// ---- 04_Application/OPC/OpcUa.TcPOU
PROGRAM OpcUa
///////////////////
// OPC UA Management 
// Commands are resetted to FALSE right after being received . Protection against rapide consecutives commands . Protection against simultaneous commands.
///////////////////
VAR_INPUT PERSISTENT
	ParamTimeOutTc			: TIME:=T#1S;		(* (s)Minimum duration before two consecutives commands *)
	ParamNbCmdBlock			: UINT  := 1 ; 		(* Number of commands per block. Commands in the same block can not be executed in the same time. *)
//Test
END_VAR             		
                    		
                    		
VAR_INPUT           		
                    		
    {attribute 'OPC.UA.DA' := '1'}                		
	AllDataR 				: AllDataR; // All Data Read Only
	
	{attribute 'OPC.UA.DA' := '1'}                		
	AllDataWPulse 			: AllDataWPulse; //  All boolean OPC UA to be written  that will be converted to tap by resetting the entry to false after two seconds. 
	
	AllDataWToggle 			: AllDataWToggle; // All boolean OPC UA to be written as a toggle
    
    {attribute 'OPC.UA.DA' := '1'}            		
	AllValueW 				: AllValueW; // All non boolean OPC UA data to be  written 
	                		
	AllRtc					: AllDataWPulse;	// OUtput of the AllDataWPulse . 
	
	// Test Mise à jour Parameters via OPC UA
	
	//AllDataParameterWrite	: AllDataParameter;	// Structure qui permet d'écrire les valeurs des paramètres via OPC UA
   		
END_VAR             		
VAR                 		
//	Buffer_AllW				: ARRAY[1..500] OF BOOL ;      
	Buffer_TcWord			: ARRAY[1..500] OF BOOL ;  
	Buffer_Rtc   			: ARRAY[1..500] OF BOOL ;  
	
	CP_TcAllow				: BOOL; // The power plan can received TC

	bInit					: BOOL;
	TempoTcRunning			: TON;
	                		
	// M_TC //      		
	TcIsRunning				: BOOL;
	NbTcAskedBlock			: BYTE;	    
	bTooManyCmd				: BOOL;		// At least one block has too many simultaneous commands. 
	bAtLeastOne				: BOOL;     // There is at least one commAND                              
	                        
	// M_ACKNOWLEDGE        
	F_Tap_OPC				: ARRAY[1..23] OF FB_TapVariable ; 
	F_Tap_OPC_SUB_MV		: ARRAY[1..16] OF FB_TapVariable ; 
	F_Tap_OPC_PTR			: ARRAY[1..CstNbPTR_G] OF ARRAY[1..6] OF FB_TapVariable ;		
	F_Tap_OPC_Inv			: ARRAY[1..CstNbPTR_G] OF ARRAY[1..CstNbInv_PTR_G] OF ARRAY[1..4] OF FB_TapVariable ;		
	F_Tap_OPC_GRID			: ARRAY[1..10] OF FB_TapVariable ; 
	F_Tap_OPC_PP			: ARRAY[1..10] OF FB_TapVariable ;	
	F_Tap_OPC_SUB_MV_InhibRead		: ARRAY[1..10] OF FB_TapVariable ;	
	
	
	F_Tap_OPC_INV_InhibRead : ARRAY[1..CstNbPTR_G] OF ARRAY[1..CstNbInv_PTR_G] OF FB_TapVariable ;	
	F_Tap_OPC_SL_InhibRead : ARRAY[1..CstNbPTR_G] OF FB_TapVariable ;	

	F_Tap_Inhib : ARRAY[1..1000] OF FB_TapVariable ;	
	
	
	Test_SmS_Rtrig			: R_TRIG ; 
	Rtrig_StayConnect		: R_TRIG;
	Rtrig_IpLauncher		: R_TRIG;
	Rtrig_HHCollector		: R_TRIG;
	Rtrig_RestartPlc		: R_TRIG;
	R_TRIGTanPhi			: R_TRIG ; 
	R_TRIG_InhibIO			: R_TRIG;
	bReadFromTargetInfos	: BOOL ; 
	// Intermediary commands
	PP_SetptP_Old							: REAL;
	PP_SetptQ_Old							: REAL;
	

	
END_VAR


VAR
	// WAGO Variable transcription
	OpcUaServer_1 : REAL ; 
	OpcUaServer_2 : REAL ; 
	OpcUaServer_3 : REAL ; 
	OpcUaServer_4 : REAL ; 
	OpcUaServer_5 : REAL ; 
	OpcUaServer_6 : REAL ; 
	OpcUaServer_7 : REAL ; 
	OpcUaServer_8 : REAL ; 
	OpcUaServer_9 : REAL ; 
	OpcUaServer_10 : REAL ; 
	OpcUaServer_11 : REAL ; 
	OpcUaServer_12 : REAL ; 
	OpcUaServer_13 : REAL ; 
	OpcUaServer_14 : REAL ; 
	OpcUaServer_15 : REAL ; 
	OpcUaServer_16 : REAL ; 
	OpcUaServer_17 : REAL ; 
	OpcUaServer_18 : REAL ; 
	OpcUaServer_19 : REAL ; 
	OpcUaServer_20 : REAL ; 
	OpcUaServer_21 : REAL ; 
	OpcUaServer_22 : REAL ; 
	OpcUaServer_23 : REAL ; 
	OpcUaServer_24 : REAL ; 
	OpcUaServer_25 : REAL ; 
	OpcUaServer_26 : REAL ; 
	OpcUaServer_27 : REAL ; 
	OpcUaServer_28 : REAL ; 
	OpcUaServer_29 : REAL ; 
	OpcUaServer_30 : REAL ; 
	OpcUaServer_31 : REAL ; 
	OpcUaServer_32 : REAL ; 
	OpcUaServer_33 : REAL ; 
	OpcUaServer_34 : REAL ; 
	OpcUaServer_35 : REAL ; 
	OpcUaServer_36 : REAL ; 
	OpcUaServer_37 : REAL ; 
	OpcUaServer_38 : REAL ; 
	OpcUaServer_39 : REAL ; 
	OpcUaServer_40 : REAL ; 
	OpcUaServer_41 : REAL ; 
	OpcUaServer_42 : REAL ; 
	OpcUaServer_43 : REAL ; 

END_VAR

	IF NOT bInit THEN
		M_Init() ; 
		bInit		:= TRUE ; 
	ELSE
		CP_TcAllow := TRUE;
		M_Evaluate();
		M_TC();
		M_Acknowledge();
		M_InhibAllowAll() ; 
		//M_Wago()
	END_IF

METHOD M_Acknowledge : BOOL
VAR
		KK: INT;
		LL: INT;
	JJ: UINT;
	TapTrigger: BOOL;
END_VAR


// 					ATTENTION				//
// Utiliser le AllRtc et pas le AllDataR 	//

	
// Defaults Actions
	// Reset SMS Server
	F_Tap_OPC[2](TapTrigger:= AllRtc.CmdReset_ServerSMS , TapOut := SMS_Server.IN_Reset_SmsServer) ; 
	// Delete all SMS
	F_Tap_OPC[3](TapTrigger:= AllRtc.CmdDeleteAllSms , TapOut := SMS_Server.IN_CmdDeleteAllSms) ; 
	// Update SMS & Mail Informations
	F_Tap_OPC[4](TapTrigger:= AllRtc.CmdChangeInfos_PhoneEmail , TapOut := SMS_Server.IN_ChangePhoneMailInfos_OPC) ; 
	F_Tap_OPC[5](TapTrigger:= AllRtc.CmdChangeInfos_PhoneEmail , TapOut := FUN_SendMail.IN_ChangePhoneMailInfos_OPC) ; 
	bReadFromTargetInfos :=	AllRtc.CmdReadInfosFromTarget_PhoneEmail ; 
	// Collect Ip Public
	Rtrig_IpLauncher(CLK:=AllRtc.CmdIpLauncher);
	F_Tap_OPC[6](TapTrigger:= Rtrig_IpLauncher.Q , TapOut := PRG_AnnexesFunctions.IN_bStart_IP) ; 
	
	// Toogle Forced Connect
	Rtrig_StayConnect(CLK:=AllRtc.CmdForcedStay_Connect);
	IF Rtrig_StayConnect.Q THEN
		A1_PP.ParamForcedStayConnect := NOT	A1_PP.ParamForcedStayConnect ;
	END_IF
	// Restart PLC
	//Rtrig_RestartPlc(CLK:=AllRtc.CmdRestart_PLC);
	F_Tap_OPC[8](TapTrigger:= AllRtc.CmdRestart_PLC , TapOut := PRG_AnnexesFunctions.IN_bStart_PLC) ; 
	// Restart Routeur ADSL
	F_Tap_OPC[9](TapTrigger:= AllRtc.CmdReset_Router_ADSL, TapOut := A1_SUBMV.A1_Router_ADSL.IN_CmdRestart) ; 
	//Reset MailServer
	F_Tap_OPC[10](TapTrigger:= AllRtc.CmdReset_ServerMail, TapOut := FUN_SendMail.IN_Reset_OPC) ; 
	// Test sms
	Test_SmS_Rtrig(CLK:=AllRtc.CmdTestSms);
	F_Tap_OPC[11](TapTrigger:= Test_SmS_Rtrig.Q, TapOut := A1_PP.IN_TestMailSms) ; 	
	// Restart Routeur 4G
	F_Tap_OPC[12](TapTrigger:= AllRtc.CmdReset_Router_4G, TapOut := A1_SUBMV.A1_Router_4G.IN_CmdRestart) ;
 	// Restart IPC
	F_Tap_OPC[13](TapTrigger:= AllRtc.CmdReset_IPC, TapOut := A1_SUBMV.A1_IPC.IN_CmdRestart) ;
	
	// Disable sms serveur
	F_Tap_OPC[14](TapTrigger:= AllDataWToggle.CmdStopServer_SMS, TapOut := FUN_Alarms.ParamDisableSMS) ; 
	// Start VPN
	F_Tap_OPC[15](TapTrigger:= AllRtc.CmdStart_Vpn, TapOut := PRG_AnnexesFunctions.IN_bStartVpnConnection) ; 
	// Stop VPN
	F_Tap_OPC[16](TapTrigger:= AllRtc.CmdStop_Vpn, TapOut := PRG_AnnexesFunctions.IN_bStopVpnConnection) ;

	
	
	// Restart Services
	F_Tap_OPC[17](TapTrigger:= AllRtc.CmdRestart_HH 		, TapOut := PRG_AnnexesFunctions.IN_CmdRestart_HH) ; // 1
	F_Tap_OPC[18](TapTrigger:= AllRtc.CmdRestart_OPCUA 		 , TapOut := PRG_AnnexesFunctions.IN_CmdRestart_OPCUA) ; // 
	F_Tap_OPC[19](TapTrigger:= AllRtc.CmdRestart_OpenVPN 	 , TapOut := PRG_AnnexesFunctions.IN_CmdRestart_OpenVPN 	 ) ; // 
	F_Tap_OPC[20](TapTrigger:= AllRtc.CmdRestart_Teamviewer	 , TapOut := PRG_AnnexesFunctions.IN_CmdRestart_Teamviewer) ; // 
	F_Tap_OPC[21](TapTrigger:= AllRtc.CmdRestart_HMIServer 	 , TapOut := PRG_AnnexesFunctions.IN_CmdRestart_HMIServer ) ; // 
	F_Tap_OPC[22](TapTrigger:= AllRtc.CmdRestart_Docker 	 , TapOut := PRG_AnnexesFunctions.IN_CmdRestart_Docker 	  ) ; // 
	F_Tap_OPC[23](TapTrigger:= AllRtc.CmdRestart_Codesys 	 , TapOut := PRG_AnnexesFunctions.IN_CmdRestart_Codesys 	 ) ; // 		
		
	

//SUB_MV
	F_Tap_OPC_SUB_MV[1](TapTrigger:= AllRtc.CmdOpen_MainMVCB , TapOut 	:= A1_SUBMV.IN_CmdOpenMainMVCB) ; 
	F_Tap_OPC_SUB_MV[2](TapTrigger:= AllRtc.CmdClose_MainMVCB , TapOut 	:= A1_SUBMV.IN_CmdCloseMainMVCB) ;
	F_Tap_OPC_SUB_MV[3](TapTrigger:= AllRtc.CmdReset_MainMVCB , TapOut 	:= A1_SUBMV.A1_MainMVCB.IN_CmdReset_L) ; 
	F_Tap_OPC_SUB_MV[4](TapTrigger:= AllRtc.CmdRestart_UPS48 , TapOut 	:= A1_SUBMV.A1_UPS_48v.IN_CmdReStartUPS) ; 	
	
	FOR KK:= 1 TO CstNbFeederMVCB_G DO 
		F_Tap_OPC_SUB_MV[4+(KK-1)*3+1](TapTrigger:= AllRtc.CmdOpen_FeederMVCB[KK] , TapOut := A1_SUBMV.IN_CmdOpenFeederMVCB[KK]) ; 
		F_Tap_OPC_SUB_MV[4+(KK-1)*3+2](TapTrigger:= AllRtc.CmdClose_FeederMVCB[KK] , TapOut := A1_SUBMV.IN_CmdCloseFeederMVCB[KK]) ; 
		F_Tap_OPC_SUB_MV[4+(KK-1)*3+3](TapTrigger:= AllRtc.CmdReset_FeederMVCB[KK] , TapOut := A1_SUBMV.AX_FeederMVCB[KK].IN_CmdReset_L) ; 

	END_FOR 	
	
// PTR 
FOR KK := 1 TO UINT_TO_INT(CstNbPTR_G) DO
	F_Tap_OPC_PTR[KK][1](TapTrigger:= AllRtc.CmdClose_PTR[KK] , TapOut := AX_PTR[KK].A1_MainMVCB_PTR.IN_CmdClose) ;
	F_Tap_OPC_PTR[KK][2](TapTrigger:= AllRtc.CmdOpen_PTR[KK] , TapOut := AX_PTR[KK].A1_MainMVCB_PTR.IN_CmdOpen) ;
	
	FOR JJ:=1 TO CstNbInv_PTR_G DO 
		F_Tap_OPC_Inv[KK][JJ][1](TapTrigger:= AllRtc.CmdStop_INV[KK][JJ] , TapOut := AX_PTR[KK].AX_INV[JJ].IN_CmdStop_Local ) ;
		F_Tap_OPC_Inv[KK][JJ][2](TapTrigger:= AllRtc.CmdStart_INV[KK][JJ] , TapOut := AX_PTR[KK].AX_INV[JJ].IN_CmdStart_Local ) ;		
		
		F_Tap_OPC_Inv[KK][JJ][3](TapTrigger:= AllRtc.CmdToggleCom_Read[KK][JJ] , TapOut := AX_PTR[KK].AX_INV[JJ].IN_CmdToggleRead ) ;
		F_Tap_OPC_Inv[KK][JJ][4](TapTrigger:= AllRtc.CmdToggleCom_Write[KK][JJ] , TapOut := AX_PTR[KK].AX_INV[JJ].IN_CmdToggleWrite ) ;		
	
		
		
		IF AllRtc.CmdStartSetptP_INV[KK][JJ] THEN 
			AX_PTR[KK].AX_INV[JJ].IN_SetptPlimit_Local :=  AllValueW.SetpP_INV[KK][JJ] ; 
		END_IF
		IF AllRtc.CmdStopSetptP_INV[KK][JJ] THEN 
			AX_PTR[KK].AX_INV[JJ].IN_SetptPlimit_Local :=  AX_PTR[KK].AX_INV[JJ].ParamPn ; 
		END_IF
		
	END_FOR
	

	

END_FOR

// DEIE
	F_Tap_OPC_GRID[1](TapTrigger:= AllRtc.CmdAutCpl , TapOut := A1_SUBMV.A1_GRID.IN_CmdAutCpl_other) ; 
	F_Tap_OPC_GRID[2](TapTrigger:= AllRtc.CmdDisconnect , TapOut := A1_SUBMV.A1_GRID.IN_CmdDisconnect_other) ; 
	F_Tap_OPC_GRID[3](TapTrigger:= AllRtc.CmdDisconnect_end , TapOut := A1_SUBMV.A1_GRID.IN_CmdDisconnect_end_other) ; 
	F_Tap_OPC_GRID[4](TapTrigger:= AllRtc.CmdEmergencyDisconnect , TapOut := A1_SUBMV.A1_GRID.IN_CmdEmergencyDisconnect_other) ; 	
	F_Tap_OPC_GRID[5](TapTrigger:= AllRtc.CmdEmergencyDisconnect_end , TapOut := A1_SUBMV.A1_GRID.IN_CmdEmergencyDisconnect_End_other) ; 	
	F_Tap_OPC_GRID[6](TapTrigger:= AllRtc.CmdStartPReg 		, TapOut := A1_SUBMV.A1_GRID.IN_CmdStartPReg_other) ; 
	F_Tap_OPC_GRID[7](TapTrigger:= AllRtc.CmdStopPReg 		, TapOut := A1_SUBMV.A1_GRID.IN_CmdStopPReg_other) ; 
	F_Tap_OPC_GRID[8](TapTrigger:= AllRtc.CmdStartQReg 		, TapOut := A1_SUBMV.A1_GRID.IN_CmdStartQReg_other) ; 
	F_Tap_OPC_GRID[9](TapTrigger:= AllRtc.CmdStopQReg 		, TapOut := A1_SUBMV.A1_GRID.IN_CmdStopQReg_other) ; 


//SUB_MV
	IF AllRtc.CmdStartLocalSetptP_PP THEN
		A1_PP.IN_PIDP_SetptP_local			:=	AllValueW.SetpP_SUB;
		A1_PP.IN_CmdPIDP_LocalMode 	:= TRUE;
	END_IF
	
	IF AllRtc.CmdStopLocalSetptP_PP THEN
		A1_PP.IN_CmdPIDP_LocalMode  	:= FALSE; 
		A1_PP.IN_PIDP_SetptP_local		:= A1_PP.ParamPmax;               
	END_IF
	
	
// PP 
	R_TRIGTanPhi(CLK:= AllRtc.CmdWriteSetptTanPhi ) ; 
	IF R_TRIGTanPhi.Q THEN 
		A1_PP.Param_SetptTanPhi  :=  AllValueW.SetptTanPhi_PP ; 		
	END_IF


//MAIL - SMS 
IF bReadFromTargetInfos THEN 
	AllValueW.AX_MailAddr_OPC		 := AllDataR.MAIL.AX_MailAddr   ; 
	AllValueW.AX_NamesUsers_OPC 	 := AllDataR.MAIL.AX_NomUtili 	; 
	AllValueW.AX_NbPhone_OPC		 := AllDataR.SMS.AX_Numtel 		; 	
	AllValueW.AX_SubscribedMail_OPC  := AllDataR.MAIL.AX_Subscribed ; 	
	AllValueW.AX_SubscribedSms_OPC   := AllDataR.SMS.AX_Subscribed  ; 	
	AllValueW.AX_UserLVL 			 := AllDataR.MAIL.AX_UserLVL    ;  		
	
	bReadFromTargetInfos 			 := FALSE ;
END_IF
END_METHOD

METHOD M_AlarmManagement
//////////////////
// Generates object alarms and manages resets. 
//////////////////

VAR 
	// Method local variables (reinitialized at each cycle) 
	FB_AlarmCodeManager			: FB_AlarmCodeManager ;

	TransfoAlarmCode			: WORD;
	TransfoWarningCode			: WORD;
	ANATempWarningCode			: WORD;    // ANA Temperature Warning Code synthesis 
	ANATempAlarmCode			: WORD;    // ANA Temperature Alarm Code synthesis                               

	AlarmCodeSD_Transfo			: WORD;    // Sd Alarm Code synthesis PTR
	AlarmCodeSD_INV				: WORD;    // Sd Alarm Code synthesis SCADA
	
	VaneWarningCode             : WORD;
	TempSensor_Amb_1WarningCode	: WORD;
	TempSensor_Amb_2WarningCode	: WORD;
	TempSensor_TransfoWarningCode: WORD;

	InvComWarning				: BOOL;		// Aggregated communication warning
	InvComError					: BOOL;		// Aggregated communication Alarm
	InvAlarmCode				: WORD; 
	InvWarningcode				: WORD;
	
	DS_Transfo					: BOOL;
	DS_INV						: BOOL;
END_VAR

	
// ALARM CODE //
	FB_AlarmCodeManager(
		bAlarm1			:= FALSE,//
		bAlarm2			:= FALSE,//
		bAlarm3			:= FALSE,//
		bAlarm4			:= FALSE,//
		bAlarm5			:= FALSE,//
		bAlarm6			:= FALSE,//
		bAlarm7			:= FALSE,//
		bAlarm8			:= FALSE,//
		bAlarm9			:= FALSE,//
		bAlarm10		:= FALSE,//
		bAlarm11		:= FALSE,//
		bAlarm12		:= FALSE,//
		bAlarm13		:= FALSE,//
		bAlarm14		:= FALSE,//
		bAlarm15		:= FALSE,//
		wAlarmCode		=> AllDataR.MesAlarmCode);

// WARNING CODE //
	FB_AlarmCodeManager(
 		bAlarm1			:= CP_TcAllow AND bTooManyCmd AND NOT   TcIsRunning,	// two many action in the same time requested                                 
		bAlarm2			:= bAtLeastOne AND  NOT bTooManyCmd AND NOT CP_TcAllow,  					// Cmd send but the PP do not allow TC
		bAlarm3			:= CP_TcAllow AND bAtLeastOne AND  NOT bTooManyCmd AND   TcIsRunning,		// Wait for previous command to be executed.
		bAlarm4			:= FALSE,//
		bAlarm5			:= FALSE,//
		bAlarm6			:= FALSE,//
		bAlarm7			:= FALSE,//
		bAlarm8			:= FALSE,//
		bAlarm9			:= FALSE,//
		bAlarm10		:= FALSE,//
		bAlarm11		:= FALSE,//
		bAlarm12		:= FALSE,//
		bAlarm13		:= FALSE,//
		bAlarm14		:= FALSE,//
        bAlarm15		:= FALSE,//
		wAlarmCode		=> AllDataR.MesWarningCode);
FB_AlarmCodeManager(
bAlarm1         :=allDataWPulse.CmdReset_ServerSMS,//Reset SMS Server #Interface
bAlarm2         :=allDataWPulse.CmdReset_ServerMail,//Reset Mail server #Interface
bAlarm3         :=allDataWPulse.CmdReset_Router_ADSL,//Restart ADSL router #Interface
bAlarm4         :=allDataWPulse.CmdReset_Router_4G,//Restart 4G router #Interface
bAlarm5         :=allDataWPulse.CmdReset_IPC,//Restart IPC #Interface
bAlarm6         :=allDataWPulse.CmdDeleteAllSms,//Delete all SMS in the buffer #Interface
bAlarm7         :=allDataWPulse.CmdChangeInfos_PhoneEmail,//Apply new changes in MAil and SMS infos #Interface
bAlarm8         :=allDataWPulse.CmdTestSms,//Test SMS function #Interface
bAlarm9         :=allDataWPulse.CmdRestart_HH,//Restart HH #Interface
bAlarm10         :=allDataWPulse.CmdRestart_OPCUA,//Restart OPCUA #Interface
bAlarm11         :=allDataWPulse.CmdRestart_OpenVPN,//Restart OpenVPN #Interface
bAlarm12         :=allDataWPulse.CmdRestart_Teamviewer,//Restart Teamviewer #Interface
bAlarm13         :=allDataWPulse.CmdRestart_HMIServer,//Restart HMIServer #Interface
bAlarm14         :=allDataWPulse.CmdRestart_Docker,//Restart Docker #Interface
bAlarm15         :=allDataWPulse.CmdRestart_Codesys,//Restart Codesys #Interface
wAlarmCode      => AllDataR.MesEventCode[1]);   
FB_AlarmCodeManager(
bAlarm1         :=allDataWPulse.CmdRestart_PLC,//Restart PLC #Interface
bAlarm2         :=allDataWPulse.CmdForcedStay_Connect,//Force the power plant to remains connected during a code restart or reboot #Interface
bAlarm3         :=allDataWPulse.CmdIpLauncher,//Get the public IP of the power plant #Interface
bAlarm4         :=allDataWPulse.CmdStart_Vpn,//Start VPN #Interface
bAlarm5         :=allDataWPulse.CmdStop_Vpn,//Stop VPN #Interface
bAlarm6         :=allDataWPulse.CmdInhibAllWrite,//Force all digital and analog output to FALSE when activated. Inhibate communication write #Interface
bAlarm7         :=allDataWPulse.CmdAllowAllWrite,//Force all digital and analog output to TRUE when activated.  Allow communication write #Interface
bAlarm8         :=allDataWPulse.CmdInhibAllRead,//Force all digital and analog input to FALSE when activated. Inhibate communication read #Interface
bAlarm9         :=allDataWPulse.CmdAllowAllRead,//Force all digital and analog input to FALSE when activated. Inhibate communication read #Interface
bAlarm10         :=allDataWPulse.CmdWriteSetptTanPhi,//PP Setpoint TanpHI #Interface
bAlarm11         :=allDataWPulse.CmdClose_MainMVCB,//Close MainMVCB #Interface
bAlarm12         :=allDataWPulse.CmdOpen_MainMVCB,//Open MainMVCB #Interface
bAlarm13         :=allDataWPulse.CmdReset_MainMVCB,//Open MainMVCB #Interface
bAlarm14         :=allDataWPulse.CmdOpen_FeederMVCB[1],//Open FeederMVCB [ARRAY](1) #Interface
bAlarm15         :=allDataWPulse.CmdOpen_FeederMVCB[2],//Open FeederMVCB [ARRAY](2) #Interface
wAlarmCode      => AllDataR.MesEventCode[2]);   
FB_AlarmCodeManager(
bAlarm1         :=allDataWPulse.CmdClose_FeederMVCB[1],//Close FeederMVCB [ARRAY](1) #Interface
bAlarm2         :=allDataWPulse.CmdClose_FeederMVCB[2],//Close FeederMVCB [ARRAY](2) #Interface
bAlarm3         :=allDataWPulse.CmdReset_FeederMVCB[1],//Close FeederMVCB [ARRAY](1) #Interface
bAlarm4         :=allDataWPulse.CmdReset_FeederMVCB[2],//Close FeederMVCB [ARRAY](2) #Interface
bAlarm5         :=allDataWPulse.CmdStartLocalSetptP_PP,//Activate local setpoint at substation #Interface
bAlarm6         :=allDataWPulse.CmdStopLocalSetptP_PP,//Desactivate local setpoint at substation #Interface
bAlarm7         :=allDataWPulse.CmdOpen_PTR[1],//Open corresponding PTR [ARRAY](1) #Interface
bAlarm8         :=allDataWPulse.CmdOpen_PTR[2],//Open corresponding PTR [ARRAY](2) #Interface
bAlarm9         :=allDataWPulse.CmdOpen_PTR[3],//Open corresponding PTR [ARRAY](3) #Interface
bAlarm10         :=allDataWPulse.CmdOpen_PTR[4],//Open corresponding PTR [ARRAY](4) #Interface
bAlarm11         :=allDataWPulse.CmdClose_PTR[1],//Close corresponding PTR [ARRAY](1) #Interface
bAlarm12         :=allDataWPulse.CmdClose_PTR[2],//Close corresponding PTR [ARRAY](2) #Interface
bAlarm13         :=allDataWPulse.CmdClose_PTR[3],//Close corresponding PTR [ARRAY](3) #Interface
bAlarm14         :=allDataWPulse.CmdClose_PTR[4],//Close corresponding PTR [ARRAY](4) #Interface
bAlarm15         :=allDataWPulse.CmdStart_INV[1][1],//Switch On inverter [ARRAY](1)(1) #Interface
wAlarmCode      => AllDataR.MesEventCode[3]);   
FB_AlarmCodeManager(
bAlarm1         :=allDataWPulse.CmdStart_INV[1][2],//Switch On inverter [ARRAY](1)(2) #Interface
bAlarm2         :=allDataWPulse.CmdStart_INV[2][1],//Switch On inverter [ARRAY](2)(1) #Interface
bAlarm3         :=allDataWPulse.CmdStart_INV[2][2],//Switch On inverter [ARRAY](2)(2) #Interface
bAlarm4         :=allDataWPulse.CmdStart_INV[3][1],//Switch On inverter [ARRAY](3)(1) #Interface
bAlarm5         :=allDataWPulse.CmdStart_INV[3][2],//Switch On inverter [ARRAY](3)(2) #Interface
bAlarm6         :=allDataWPulse.CmdStart_INV[4][1],//Switch On inverter [ARRAY](4)(1) #Interface
bAlarm7         :=allDataWPulse.CmdStart_INV[4][2],//Switch On inverter [ARRAY](4)(2) #Interface
bAlarm8         :=allDataWPulse.CmdStop_INV[1][1],//Switch Off inverter [ARRAY](1)(1) #Interface
bAlarm9         :=allDataWPulse.CmdStop_INV[1][2],//Switch Off inverter [ARRAY](1)(2) #Interface
bAlarm10         :=allDataWPulse.CmdStop_INV[2][1],//Switch Off inverter [ARRAY](2)(1) #Interface
bAlarm11         :=allDataWPulse.CmdStop_INV[2][2],//Switch Off inverter [ARRAY](2)(2) #Interface
bAlarm12         :=allDataWPulse.CmdStop_INV[3][1],//Switch Off inverter [ARRAY](3)(1) #Interface
bAlarm13         :=allDataWPulse.CmdStop_INV[3][2],//Switch Off inverter [ARRAY](3)(2) #Interface
bAlarm14         :=allDataWPulse.CmdStop_INV[4][1],//Switch Off inverter [ARRAY](4)(1) #Interface
bAlarm15         :=allDataWPulse.CmdStop_INV[4][2],//Switch Off inverter [ARRAY](4)(2) #Interface
wAlarmCode      => AllDataR.MesEventCode[4]);   

FB_AlarmCodeManager(
bAlarm1         :=allDataWPulse.CmdStartSetptP_INV[1][1],//Activate local setpoint on inverter [ARRAY](1)(1) #Interface
bAlarm2         :=allDataWPulse.CmdStartSetptP_INV[1][2],//Activate local setpoint on inverter [ARRAY](1)(2) #Interface
bAlarm3         :=allDataWPulse.CmdStartSetptP_INV[2][1],//Activate local setpoint on inverter [ARRAY](2)(1) #Interface
bAlarm4         :=allDataWPulse.CmdStartSetptP_INV[2][2],//Activate local setpoint on inverter [ARRAY](2)(2) #Interface
bAlarm5         :=allDataWPulse.CmdStartSetptP_INV[3][1],//Activate local setpoint on inverter [ARRAY](3)(1) #Interface
bAlarm6         :=allDataWPulse.CmdStartSetptP_INV[3][2],//Activate local setpoint on inverter [ARRAY](3)(2) #Interface
bAlarm7         :=allDataWPulse.CmdStartSetptP_INV[4][1],//Activate local setpoint on inverter [ARRAY](4)(1) #Interface
bAlarm8         :=allDataWPulse.CmdStartSetptP_INV[4][2],//Activate local setpoint on inverter [ARRAY](4)(2) #Interface
bAlarm9         :=allDataWPulse.CmdStopSetptP_INV[1][1],//Desactivate local setpoint on inverter [ARRAY](1)(1) #Interface
bAlarm10         :=allDataWPulse.CmdStopSetptP_INV[1][2],//Desactivate local setpoint on inverter [ARRAY](1)(2) #Interface
bAlarm11         :=allDataWPulse.CmdStopSetptP_INV[2][1],//Desactivate local setpoint on inverter [ARRAY](2)(1) #Interface
bAlarm12         :=allDataWPulse.CmdStopSetptP_INV[2][2],//Desactivate local setpoint on inverter [ARRAY](2)(2) #Interface
bAlarm13         :=allDataWPulse.CmdStopSetptP_INV[3][1],//Desactivate local setpoint on inverter [ARRAY](3)(1) #Interface
bAlarm14         :=allDataWPulse.CmdStopSetptP_INV[3][2],//Desactivate local setpoint on inverter [ARRAY](3)(2) #Interface
bAlarm15         :=allDataWPulse.CmdStopSetptP_INV[4][1],//Desactivate local setpoint on inverter [ARRAY](4)(1) #Interface
wAlarmCode      => AllDataR.MesEventCode[5]);   

FB_AlarmCodeManager(
bAlarm1         :=allDataWPulse.CmdStopSetptP_INV[4][2],//Desactivate local setpoint on inverter [ARRAY](4)(2) #Interface
bAlarm2         :=allDataWPulse.CmdToggleCom_Read[1][1],//Inverter Toggle Read Communcation [ARRAY](1)(1) #Interface
bAlarm3         :=allDataWPulse.CmdToggleCom_Read[1][2],//Inverter Toggle Read Communcation [ARRAY](1)(2) #Interface
bAlarm4         :=allDataWPulse.CmdToggleCom_Read[2][1],//Inverter Toggle Read Communcation [ARRAY](2)(1) #Interface
bAlarm5         :=allDataWPulse.CmdToggleCom_Read[2][2],//Inverter Toggle Read Communcation [ARRAY](2)(2) #Interface
bAlarm6         :=allDataWPulse.CmdToggleCom_Read[3][1],//Inverter Toggle Read Communcation [ARRAY](3)(1) #Interface
bAlarm7         :=allDataWPulse.CmdToggleCom_Read[3][2],//Inverter Toggle Read Communcation [ARRAY](3)(2) #Interface
bAlarm8         :=allDataWPulse.CmdToggleCom_Read[4][1],//Inverter Toggle Read Communcation [ARRAY](4)(1) #Interface
bAlarm9         :=allDataWPulse.CmdToggleCom_Read[4][2],//Inverter Toggle Read Communcation [ARRAY](4)(2) #Interface
bAlarm10         :=allDataWPulse.CmdToggleCom_Write[1][1],//Inverter Toggle Write Communcation [ARRAY](1)(1) #Interface
bAlarm11         :=allDataWPulse.CmdToggleCom_Write[1][2],//Inverter Toggle Write Communcation [ARRAY](1)(2) #Interface
bAlarm12         :=allDataWPulse.CmdToggleCom_Write[2][1],//Inverter Toggle Write Communcation [ARRAY](2)(1) #Interface
bAlarm13         :=allDataWPulse.CmdToggleCom_Write[2][2],//Inverter Toggle Write Communcation [ARRAY](2)(2) #Interface
bAlarm14         :=allDataWPulse.CmdToggleCom_Write[3][1],//Inverter Toggle Write Communcation [ARRAY](3)(1) #Interface
bAlarm15         :=allDataWPulse.CmdToggleCom_Write[3][2],//Inverter Toggle Write Communcation [ARRAY](3)(2) #Interface
wAlarmCode      => AllDataR.MesEventCode[6]);   
FB_AlarmCodeManager(
bAlarm1         :=allDataWPulse.CmdToggleCom_Write[4][1],//Inverter Toggle Write Communcation [ARRAY](4)(1) #Interface
bAlarm2         :=allDataWPulse.CmdToggleCom_Write[4][2],//Inverter Toggle Write Communcation [ARRAY](4)(2) #Interface
bAlarm3         :=allDataWPulse.CmdRestart_UPS48,//Restart UPS #Interface
bAlarm4         :=allDataWPulse.CmdAutCpl,//Coupling authorization #Interface
bAlarm5         :=allDataWPulse.CmdDisconnect,//Powerplant disconnect order #Interface
bAlarm6         :=allDataWPulse.CmdEmergencyDisconnect,//Powerplant Emergency disconnect order #Interface
bAlarm7         :=allDataWPulse.CmdDisconnect_end,//Powerplant disconnect order #Interface
bAlarm8         :=allDataWPulse.CmdEmergencyDisconnect_end,//Powerplant Emergency disconnect order #Interface
bAlarm9         :=allDataWPulse.CmdStartPReg,//Activate P regulation from Grid #Interface
bAlarm10         :=allDataWPulse.CmdStopPreg,//Desactivate P regulation from Grid #Interface
bAlarm11         :=allDataWPulse.CmdStartQReg,//Activate Q regulation from Grid #Interface
bAlarm12         :=allDataWPulse.CmdStopQReg,//Desactivate Q regulation from Grid #Interface
bAlarm13         :=allDataWToggle.CmdStopServer_SMS,//Disable SMS Server #Interface
bAlarm14         :=allValueW.AX_SubscribedSms_OPC[1],//List of subscription for SMS function(1) #Interface
bAlarm15         :=allValueW.AX_SubscribedSms_OPC[2],//List of subscription for SMS function(2) #Interface
wAlarmCode      => AllDataR.MesEventCode[7]);   
FB_AlarmCodeManager(
bAlarm1         :=allValueW.AX_SubscribedSms_OPC[3],//List of subscription for SMS function(3) #Interface
bAlarm2         :=allValueW.AX_SubscribedSms_OPC[4],//List of subscription for SMS function(4) #Interface
bAlarm3         :=allValueW.AX_SubscribedSms_OPC[5],//List of subscription for SMS function(5) #Interface
bAlarm4         :=allValueW.AX_SubscribedSms_OPC[6],//List of subscription for SMS function(6) #Interface
bAlarm5         :=allValueW.AX_SubscribedSms_OPC[7],//List of subscription for SMS function(7) #Interface
bAlarm6         :=allValueW.AX_SubscribedSms_OPC[8],//List of subscription for SMS function(8) #Interface
bAlarm7         :=allValueW.AX_SubscribedSms_OPC[9],//List of subscription for SMS function(9) #Interface
bAlarm8         :=allValueW.AX_SubscribedSms_OPC[10],//List of subscription for SMS function(10) #Interface
bAlarm9         :=allValueW.AX_SubscribedMail_OPC[1],//List of subscription fro MAIL function(1) #Interface
bAlarm10         :=allValueW.AX_SubscribedMail_OPC[2],//List of subscription fro MAIL function(2) #Interface
bAlarm11         :=allValueW.AX_SubscribedMail_OPC[3],//List of subscription fro MAIL function(3) #Interface
bAlarm12         :=allValueW.AX_SubscribedMail_OPC[4],//List of subscription fro MAIL function(4) #Interface
bAlarm13         :=allValueW.AX_SubscribedMail_OPC[5],//List of subscription fro MAIL function(5) #Interface
bAlarm14         :=allValueW.AX_SubscribedMail_OPC[6],//List of subscription fro MAIL function(6) #Interface
bAlarm15         :=allValueW.AX_SubscribedMail_OPC[7],//List of subscription fro MAIL function(7) #Interface
wAlarmCode      => AllDataR.MesEventCode[8]);   
FB_AlarmCodeManager(
bAlarm1         :=allValueW.AX_SubscribedMail_OPC[8],//List of subscription fro MAIL function(8) #Interface
bAlarm2         :=allValueW.AX_SubscribedMail_OPC[9],//List of subscription fro MAIL function(9) #Interface
bAlarm3         :=allValueW.AX_SubscribedMail_OPC[10],//List of subscription fro MAIL function(10) #Interface
wAlarmCode      => AllDataR.MesEventCode[9]);
END_METHOD

METHOD M_Evaluate : BOOL
VAR_INPUT
END_VAR


VAR
	KK: UINT;
END_VAR

AllDataR.PP			:=  A1_PP.MesData ; 
AllDataR.SUBMV	    :=  A1_SUBMV.MesDataExd; 
FOR KK:=1 TO CstNbPTR_G DO
	AllDataR.PTR[KK]	    :=  AX_PTR[KK].MesDataExd;
END_FOR


AllDataR.WS	        :=  A1_WS.MesDataExd; 

AllDataR.SMS	    :=  SMS_Server.MesData;
AllDataR.MAIL       :=  FUN_SendMail.MesData;

AllDataR.CSV		:= FUN_Alarms_CSV.MesData; 
AllDataR.CSVData := FUN_Write_CSV.WriteValue.MesData ;
END_METHOD

METHOD M_InhibAllowAll : BOOL
VAR
		KK: INT;
		LL: INT;
	JJ: UINT;
	TapTrigger: BOOL;
END_VAR


// 					ATTENTION				//
// Utiliser le AllRtc et pas le AllDataR 	//
// Inhib all write 
	// Inhib IO 
	IF AllRtc.CmdInhibAllWrite THEN 
		PRG_IO.IN_CmdInhibOutput_OPC :=  TRUE ;  // Toggle the command for output . 
	ELSIF AllRtc.CmdAllowAllWrite THEN 
		PRG_IO.IN_CmdInhibOutput_OPC :=  FALSE ;  // Toggle the command for output . 
	END_IF 
	
	// Inhib Com
END_METHOD

METHOD M_Init : BOOL
VAR_INPUT
END_VAR
																
//AllDataWPulse.CmdInhibAllWrite := TRUE  	;
END_METHOD

METHOD M_TC : BOOL
VAR_INPUT
END_VAR

VAR
	AllDataW_0 				: AllDataWPulse; // All Data Write
	KK						: UINT;
	BlockElemCount			: UINT;	// Current element in current block.

END_VAR
MEMCPY(srcAddr := ADR(AllDataWPulse) ,destAddr:= ADR(Buffer_TcWord) ,n:= SIZEOF(AllDataWPulse) ) ; 

NbTcAskedBlock	:= 0;
TcIsRunning		:= FALSE ; 
BlockElemCount 	:=1 ;
bTooManyCmd 	:= FALSE ; 
bAtLeastOne		:= FALSE ;

FOR KK:=1 TO SIZEOF(AllDataWPulse) DO 
	
	IF Buffer_TcWord[KK] THEN // la commande est à True . 
		NbTcAskedBlock := NbTcAskedBlock + 1 ; 
	END_IF
	
	IF Buffer_Rtc[KK] THEN // une commande est en cours 
		TcIsRunning:= TRUE   ;
	END_IF	
	
	IF ParamNbCmdBlock <= BlockElemCount THEN // Fin d'un block. On regarde si il y a eu une commande mais pas plusieurs. 
		BlockElemCount := 1 ; 
		bTooManyCmd	:=bTooManyCmd  OR  NbTcAskedBlock>1 ; 
		bAtLeastOne :=bAtLeastOne  OR NbTcAskedBlock=1; 
		NbTcAskedBlock := 0 ;
		
	ELSE
		BlockElemCount :=  BlockElemCount + 1 ;
	END_IF
END_FOR
// To consider last block
bAtLeastOne := bAtLeastOne OR  NbTcAskedBlock=1; 	
bTooManyCmd	:= bTooManyCmd OR  NbTcAskedBlock>1 ; 

IF CP_TcAllow AND bAtLeastOne AND NOT bTooManyCmd AND NOT TcIsRunning THEN 	// On ne process les commandes que si aucun block n'a pas de double commande, mais qu'au moins un en a une. 
	Buffer_Rtc := Buffer_TcWord  ; 
END_IF

MEMCPY(srcAddr := ADR(Buffer_Rtc) ,destAddr:= ADR(AllRtc) ,n:= SIZEOF(AllRtc) ) ; 

IF bAtLeastOne OR bTooManyCmd THEN 
	//Reset at each cycle
	AllDataWPulse := AllDataW_0;
END_IF


//SECURITY
	TempoTcRunning(IN:= TcIsRunning AND CP_TcAllow , PT:=ParamTimeOutTc);
	
	IF TempoTcRunning.Q THEN
		AllRtc 	:= AllDataW_0;
		FOR KK:= 1 TO SIZEOF(AllDataWPulse) DO 
			Buffer_Rtc[KK]	:= FALSE;
		END_FOR 
	END_IF
END_METHOD

METHOD M_UpdateParameters : BOOL
VAR_INPUT
END_VAR
(*
// Update Parameters
FB_WriteOnChange[1](VarInput := ADR(AllDataParameterWrite.PP_ParamPmax) , VarOut := ADR(A1_PP.ParamPmax), Size:=SIZEOF(A1_PP.ParamPmax) ); 
FB_WriteOnChange[2](VarInput := ADR(AllDataParameterWrite.PP_ParamPmin) , VarOut := ADR(A1_PP.ParamPmin), Size:=SIZEOF(A1_PP.ParamPmin) ); 
FB_WriteOnChange[3](VarInput := ADR(AllDataParameterWrite.PP_ParamQmax) , VarOut := ADR(A1_PP.ParamQmax), Size:=SIZEOF(A1_PP.ParamQmax) ); 
FB_WriteOnChange[4](VarInput := ADR(AllDataParameterWrite.PP_ParamQmin) , VarOut := ADR(A1_PP.ParamQmin), Size:=SIZEOF(A1_PP.ParamQmin) ); 
FB_WriteOnChange[5](VarInput := ADR(AllDataParameterWrite.PP_ParamNominalVoltage) , VarOut := ADR(A1_PP.ParamNominalVoltage), Size:=SIZEOF(A1_PP.ParamNominalVoltage) ); 
FB_WriteOnChange[6](VarInput := ADR(AllDataParameterWrite.PP_ParamNominalFrequency) , VarOut := ADR(A1_PP.ParamNominalFrequency), Size:=SIZEOF(A1_PP.ParamNominalFrequency) ); 
FB_WriteOnChange[7](VarInput := ADR(AllDataParameterWrite.PP_ParamQmaxPbelow20) , VarOut := ADR(A1_PP.ParamQmaxPbelow20), Size:=SIZEOF(A1_PP.ParamQmaxPbelow20) ); 
FB_WriteOnChange[8](VarInput := ADR(AllDataParameterWrite.PP_ParamTanPhiMax) , VarOut := ADR(A1_PP.ParamTanPhiMax), Size:=SIZEOF(A1_PP.ParamTanPhiMax) ); 
FB_WriteOnChange[9](VarInput := ADR(AllDataParameterWrite.PP_ParamTanPhiMin) , VarOut := ADR(A1_PP.ParamTanPhiMin), Size:=SIZEOF(A1_PP.ParamTanPhiMin) ); 
FB_WriteOnChange[10](VarInput := ADR(AllDataParameterWrite.PP_ParamLocalMode) , VarOut := ADR(A1_PP.ParamLocalMode), Size:=SIZEOF(A1_PP.ParamLocalMode) ); 
FB_WriteOnChange[11](VarInput := ADR(AllDataParameterWrite.PP_ParamQcontrol) , VarOut := ADR(A1_PP.ParamQcontrol), Size:=SIZEOF(A1_PP.ParamQcontrol) ); 
FB_WriteOnChange[12](VarInput := ADR(AllDataParameterWrite.PP_ParamTanPhiCtrl) , VarOut := ADR(A1_PP.ParamTanPhiCtrl), Size:=SIZEOF(A1_PP.ParamTanPhiCtrl) ); 
FB_WriteOnChange[13](VarInput := ADR(AllDataParameterWrite.PP_Param_SetptTanPhi) , VarOut := ADR(A1_PP.Param_SetptTanPhi), Size:=SIZEOF(A1_PP.Param_SetptTanPhi) ); 
FB_WriteOnChange[14](VarInput := ADR(AllDataParameterWrite.PP_ParamPoffset_OL) , VarOut := ADR(A1_PP.ParamPoffset_OL), Size:=SIZEOF(A1_PP.ParamPoffset_OL) ); 
FB_WriteOnChange[15](VarInput := ADR(AllDataParameterWrite.PP_ParamQoffset_OL) , VarOut := ADR(A1_PP.ParamQoffset_OL), Size:=SIZEOF(A1_PP.ParamQoffset_OL) ); 
FB_WriteOnChange[16](VarInput := ADR(AllDataParameterWrite.PP_ParamPIDP_K) , VarOut := ADR(A1_PP.ParamPIDP_K), Size:=SIZEOF(A1_PP.ParamPIDP_K) ); 
FB_WriteOnChange[17](VarInput := ADR(AllDataParameterWrite.PP_ParamPidP_I) , VarOut := ADR(A1_PP.ParamPidP_I), Size:=SIZEOF(A1_PP.ParamPidP_I) ); 
FB_WriteOnChange[18](VarInput := ADR(AllDataParameterWrite.PP_ParamPidP_D) , VarOut := ADR(A1_PP.ParamPidP_D), Size:=SIZEOF(A1_PP.ParamPidP_D) ); 
FB_WriteOnChange[19](VarInput := ADR(AllDataParameterWrite.PP_ParamPIDQ_K) , VarOut := ADR(A1_PP.ParamPIDQ_K), Size:=SIZEOF(A1_PP.ParamPIDQ_K) ); 
FB_WriteOnChange[20](VarInput := ADR(AllDataParameterWrite.PP_ParamPidQ_I) , VarOut := ADR(A1_PP.ParamPidQ_I), Size:=SIZEOF(A1_PP.ParamPidQ_I) ); 
FB_WriteOnChange[21](VarInput := ADR(AllDataParameterWrite.PP_ParamPidQ_D) , VarOut := ADR(A1_PP.ParamPidQ_D), Size:=SIZEOF(A1_PP.ParamPidQ_D) ); 
FB_WriteOnChange[22](VarInput := ADR(AllDataParameterWrite.PP_ParamPIDQMin) , VarOut := ADR(A1_PP.ParamPIDQMin), Size:=SIZEOF(A1_PP.ParamPIDQMin) ); 
FB_WriteOnChange[23](VarInput := ADR(AllDataParameterWrite.PP_ParamPIDQMax) , VarOut := ADR(A1_PP.ParamPIDQMax), Size:=SIZEOF(A1_PP.ParamPIDQMax) ); 
FB_WriteOnChange[24](VarInput := ADR(AllDataParameterWrite.PP_ParamQfUQmin) , VarOut := ADR(A1_PP.ParamQfUQmin), Size:=SIZEOF(A1_PP.ParamQfUQmin) ); 
FB_WriteOnChange[25](VarInput := ADR(AllDataParameterWrite.PP_ParamQfUQmax) , VarOut := ADR(A1_PP.ParamQfUQmax), Size:=SIZEOF(A1_PP.ParamQfUQmax) ); 
FB_WriteOnChange[26](VarInput := ADR(AllDataParameterWrite.PP_ParamQfUUHigh) , VarOut := ADR(A1_PP.ParamQfUUHigh), Size:=SIZEOF(A1_PP.ParamQfUUHigh) ); 
FB_WriteOnChange[27](VarInput := ADR(AllDataParameterWrite.PP_ParamQfUDdBandHigh) , VarOut := ADR(A1_PP.ParamQfUDdBandHigh), Size:=SIZEOF(A1_PP.ParamQfUDdBandHigh) ); 
FB_WriteOnChange[28](VarInput := ADR(AllDataParameterWrite.PP_ParamQfUDdBandLow) , VarOut := ADR(A1_PP.ParamQfUDdBandLow), Size:=SIZEOF(A1_PP.ParamQfUDdBandLow) ); 
FB_WriteOnChange[29](VarInput := ADR(AllDataParameterWrite.PP_ParamQfUULow) , VarOut := ADR(A1_PP.ParamQfUULow), Size:=SIZEOF(A1_PP.ParamQfUULow) ); 
FB_WriteOnChange[30](VarInput := ADR(AllDataParameterWrite.PP_ParamNofeedingTime) , VarOut := ADR(A1_PP.ParamNofeedingTime), Size:=SIZEOF(A1_PP.ParamNofeedingTime) ); 
FB_WriteOnChange[31](VarInput := ADR(AllDataParameterWrite.PP_ParamNofeedingWarningTime) , VarOut := ADR(A1_PP.ParamNofeedingWarningTime), Size:=SIZEOF(A1_PP.ParamNofeedingWarningTime) ); 
FB_WriteOnChange[32](VarInput := ADR(AllDataParameterWrite.PP_ParamNofeedingAlarmTime) , VarOut := ADR(A1_PP.ParamNofeedingAlarmTime), Size:=SIZEOF(A1_PP.ParamNofeedingAlarmTime) ); 
FB_WriteOnChange[33](VarInput := ADR(AllDataParameterWrite.PP_ParamDiscoAlarmTime) , VarOut := ADR(A1_PP.ParamDiscoAlarmTime), Size:=SIZEOF(A1_PP.ParamDiscoAlarmTime) ); 
FB_WriteOnChange[34](VarInput := ADR(AllDataParameterWrite.PP_ParamForcedStayConnect) , VarOut := ADR(A1_PP.ParamForcedStayConnect), Size:=SIZEOF(A1_PP.ParamForcedStayConnect) ); 
FB_WriteOnChange[35](VarInput := ADR(AllDataParameterWrite.PP_ParamMinimalDiskSpace) , VarOut := ADR(A1_PP.ParamMinimalDiskSpace), Size:=SIZEOF(A1_PP.ParamMinimalDiskSpace) ); 
FB_WriteOnChange[36](VarInput := ADR(AllDataParameterWrite.PP_ParamCodeVersion) , VarOut := ADR(A1_PP.ParamCodeVersion), Size:=SIZEOF(A1_PP.ParamCodeVersion) ); 
FB_WriteOnChange[37](VarInput := ADR(AllDataParameterWrite.PP_ParamNbCoupler) , VarOut := ADR(A1_PP.ParamNbCoupler), Size:=SIZEOF(A1_PP.ParamNbCoupler) ); 
FB_WriteOnChange[38](VarInput := ADR(AllDataParameterWrite.PTR_1_ParamPTRVersion) , VarOut := ADR(AX_PTR[1].ParamPTRVersion), Size:=SIZEOF(AX_PTR[1].ParamPTRVersion) ); 
FB_WriteOnChange[39](VarInput := ADR(AllDataParameterWrite.PTR_2_ParamPTRVersion) , VarOut := ADR(AX_PTR[2].ParamPTRVersion), Size:=SIZEOF(AX_PTR[2].ParamPTRVersion) ); 
FB_WriteOnChange[40](VarInput := ADR(AllDataParameterWrite.PTR_3_ParamPTRVersion) , VarOut := ADR(AX_PTR[3].ParamPTRVersion), Size:=SIZEOF(AX_PTR[3].ParamPTRVersion) ); 
FB_WriteOnChange[41](VarInput := ADR(AllDataParameterWrite.PTR_4_ParamPTRVersion) , VarOut := ADR(AX_PTR[4].ParamPTRVersion), Size:=SIZEOF(AX_PTR[4].ParamPTRVersion) ); 
FB_WriteOnChange[42](VarInput := ADR(AllDataParameterWrite.PTR_1_ParamTimeOutStart) , VarOut := ADR(AX_PTR[1].ParamTimeOutStart), Size:=SIZEOF(AX_PTR[1].ParamTimeOutStart) ); 
FB_WriteOnChange[43](VarInput := ADR(AllDataParameterWrite.PTR_2_ParamTimeOutStart) , VarOut := ADR(AX_PTR[2].ParamTimeOutStart), Size:=SIZEOF(AX_PTR[2].ParamTimeOutStart) ); 
FB_WriteOnChange[44](VarInput := ADR(AllDataParameterWrite.PTR_3_ParamTimeOutStart) , VarOut := ADR(AX_PTR[3].ParamTimeOutStart), Size:=SIZEOF(AX_PTR[3].ParamTimeOutStart) ); 
FB_WriteOnChange[45](VarInput := ADR(AllDataParameterWrite.PTR_4_ParamTimeOutStart) , VarOut := ADR(AX_PTR[4].ParamTimeOutStart), Size:=SIZEOF(AX_PTR[4].ParamTimeOutStart) ); 
FB_WriteOnChange[46](VarInput := ADR(AllDataParameterWrite.PTR_1_ParamTimeOutStop) , VarOut := ADR(AX_PTR[1].ParamTimeOutStop), Size:=SIZEOF(AX_PTR[1].ParamTimeOutStop) ); 
FB_WriteOnChange[47](VarInput := ADR(AllDataParameterWrite.PTR_2_ParamTimeOutStop) , VarOut := ADR(AX_PTR[2].ParamTimeOutStop), Size:=SIZEOF(AX_PTR[2].ParamTimeOutStop) ); 
FB_WriteOnChange[48](VarInput := ADR(AllDataParameterWrite.PTR_3_ParamTimeOutStop) , VarOut := ADR(AX_PTR[3].ParamTimeOutStop), Size:=SIZEOF(AX_PTR[3].ParamTimeOutStop) ); 
FB_WriteOnChange[49](VarInput := ADR(AllDataParameterWrite.PTR_4_ParamTimeOutStop) , VarOut := ADR(AX_PTR[4].ParamTimeOutStop), Size:=SIZEOF(AX_PTR[4].ParamTimeOutStop) ); 
FB_WriteOnChange[50](VarInput := ADR(AllDataParameterWrite.PTR_1_ParamTimeOutDisconnect) , VarOut := ADR(AX_PTR[1].ParamTimeOutDisconnect), Size:=SIZEOF(AX_PTR[1].ParamTimeOutDisconnect) ); 
FB_WriteOnChange[51](VarInput := ADR(AllDataParameterWrite.PTR_2_ParamTimeOutDisconnect) , VarOut := ADR(AX_PTR[2].ParamTimeOutDisconnect), Size:=SIZEOF(AX_PTR[2].ParamTimeOutDisconnect) ); 
FB_WriteOnChange[52](VarInput := ADR(AllDataParameterWrite.PTR_3_ParamTimeOutDisconnect) , VarOut := ADR(AX_PTR[3].ParamTimeOutDisconnect), Size:=SIZEOF(AX_PTR[3].ParamTimeOutDisconnect) ); 
FB_WriteOnChange[53](VarInput := ADR(AllDataParameterWrite.PTR_4_ParamTimeOutDisconnect) , VarOut := ADR(AX_PTR[4].ParamTimeOutDisconnect), Size:=SIZEOF(AX_PTR[4].ParamTimeOutDisconnect) ); 
FB_WriteOnChange[54](VarInput := ADR(AllDataParameterWrite.PTR_1_ParamTempoComAlarm) , VarOut := ADR(AX_PTR[1].ParamTempoComAlarm), Size:=SIZEOF(AX_PTR[1].ParamTempoComAlarm) ); 
FB_WriteOnChange[55](VarInput := ADR(AllDataParameterWrite.PTR_2_ParamTempoComAlarm) , VarOut := ADR(AX_PTR[2].ParamTempoComAlarm), Size:=SIZEOF(AX_PTR[2].ParamTempoComAlarm) ); 
FB_WriteOnChange[56](VarInput := ADR(AllDataParameterWrite.PTR_3_ParamTempoComAlarm) , VarOut := ADR(AX_PTR[3].ParamTempoComAlarm), Size:=SIZEOF(AX_PTR[3].ParamTempoComAlarm) ); 
FB_WriteOnChange[57](VarInput := ADR(AllDataParameterWrite.PTR_4_ParamTempoComAlarm) , VarOut := ADR(AX_PTR[4].ParamTempoComAlarm), Size:=SIZEOF(AX_PTR[4].ParamTempoComAlarm) ); 
FB_WriteOnChange[58](VarInput := ADR(AllDataParameterWrite.PTR_1_ParamTempoStartInv) , VarOut := ADR(AX_PTR[1].ParamTempoStartInv), Size:=SIZEOF(AX_PTR[1].ParamTempoStartInv) ); 
FB_WriteOnChange[59](VarInput := ADR(AllDataParameterWrite.PTR_2_ParamTempoStartInv) , VarOut := ADR(AX_PTR[2].ParamTempoStartInv), Size:=SIZEOF(AX_PTR[2].ParamTempoStartInv) ); 
FB_WriteOnChange[60](VarInput := ADR(AllDataParameterWrite.PTR_3_ParamTempoStartInv) , VarOut := ADR(AX_PTR[3].ParamTempoStartInv), Size:=SIZEOF(AX_PTR[3].ParamTempoStartInv) ); 
FB_WriteOnChange[61](VarInput := ADR(AllDataParameterWrite.PTR_4_ParamTempoStartInv) , VarOut := ADR(AX_PTR[4].ParamTempoStartInv), Size:=SIZEOF(AX_PTR[4].ParamTempoStartInv) ); 
FB_WriteOnChange[62](VarInput := ADR(AllDataParameterWrite.PTR_1_ParamTempoStopInv) , VarOut := ADR(AX_PTR[1].ParamTempoStopInv), Size:=SIZEOF(AX_PTR[1].ParamTempoStopInv) ); 
FB_WriteOnChange[63](VarInput := ADR(AllDataParameterWrite.PTR_2_ParamTempoStopInv) , VarOut := ADR(AX_PTR[2].ParamTempoStopInv), Size:=SIZEOF(AX_PTR[2].ParamTempoStopInv) ); 
FB_WriteOnChange[64](VarInput := ADR(AllDataParameterWrite.PTR_3_ParamTempoStopInv) , VarOut := ADR(AX_PTR[3].ParamTempoStopInv), Size:=SIZEOF(AX_PTR[3].ParamTempoStopInv) ); 
FB_WriteOnChange[65](VarInput := ADR(AllDataParameterWrite.PTR_4_ParamTempoStopInv) , VarOut := ADR(AX_PTR[4].ParamTempoStopInv), Size:=SIZEOF(AX_PTR[4].ParamTempoStopInv) ); 
FB_WriteOnChange[66](VarInput := ADR(AllDataParameterWrite.PTR_1_ParamPTRNum) , VarOut := ADR(AX_PTR[1].ParamPTRNum), Size:=SIZEOF(AX_PTR[1].ParamPTRNum) ); 
FB_WriteOnChange[67](VarInput := ADR(AllDataParameterWrite.PTR_2_ParamPTRNum) , VarOut := ADR(AX_PTR[2].ParamPTRNum), Size:=SIZEOF(AX_PTR[2].ParamPTRNum) ); 
FB_WriteOnChange[68](VarInput := ADR(AllDataParameterWrite.PTR_3_ParamPTRNum) , VarOut := ADR(AX_PTR[3].ParamPTRNum), Size:=SIZEOF(AX_PTR[3].ParamPTRNum) ); 
FB_WriteOnChange[69](VarInput := ADR(AllDataParameterWrite.PTR_4_ParamPTRNum) , VarOut := ADR(AX_PTR[4].ParamPTRNum), Size:=SIZEOF(AX_PTR[4].ParamPTRNum) ); 
FB_WriteOnChange[70](VarInput := ADR(AllDataParameterWrite.PTR_1_ParamNbINV) , VarOut := ADR(AX_PTR[1].ParamNbINV), Size:=SIZEOF(AX_PTR[1].ParamNbINV) ); 
FB_WriteOnChange[71](VarInput := ADR(AllDataParameterWrite.PTR_2_ParamNbINV) , VarOut := ADR(AX_PTR[2].ParamNbINV), Size:=SIZEOF(AX_PTR[2].ParamNbINV) ); 
FB_WriteOnChange[72](VarInput := ADR(AllDataParameterWrite.PTR_3_ParamNbINV) , VarOut := ADR(AX_PTR[3].ParamNbINV), Size:=SIZEOF(AX_PTR[3].ParamNbINV) ); 
FB_WriteOnChange[73](VarInput := ADR(AllDataParameterWrite.PTR_4_ParamNbINV) , VarOut := ADR(AX_PTR[4].ParamNbINV), Size:=SIZEOF(AX_PTR[4].ParamNbINV) ); 
FB_WriteOnChange[74](VarInput := ADR(AllDataParameterWrite.SUBMV_ParamTempoPoste) , VarOut := ADR(A1_SUBMV.ParamTempoPoste), Size:=SIZEOF(A1_SUBMV.ParamTempoPoste) ); 
FB_WriteOnChange[75](VarInput := ADR(AllDataParameterWrite.SUBMV_ParamTempoUnknowFault) , VarOut := ADR(A1_SUBMV.ParamTempoUnknowFault), Size:=SIZEOF(A1_SUBMV.ParamTempoUnknowFault) ); 
FB_WriteOnChange[76](VarInput := ADR(AllDataParameterWrite.SUBMV_ParamTempoSepamCloseAfterGte) , VarOut := ADR(A1_SUBMV.ParamTempoSepamCloseAfterGte), Size:=SIZEOF(A1_SUBMV.ParamTempoSepamCloseAfterGte) ); 
FB_WriteOnChange[77](VarInput := ADR(AllDataParameterWrite.SUBMV_ParamAutoCloseMainMVCBEnabled) , VarOut := ADR(A1_SUBMV.ParamAutoCloseMainMVCBEnabled), Size:=SIZEOF(A1_SUBMV.ParamAutoCloseMainMVCBEnabled) ); 
FB_WriteOnChange[78](VarInput := ADR(AllDataParameterWrite.SUBMV_ParamSUB_MVVersion) , VarOut := ADR(A1_SUBMV.ParamSUB_MVVersion), Size:=SIZEOF(A1_SUBMV.ParamSUB_MVVersion) ); 
FB_WriteOnChange[79](VarInput := ADR(AllDataParameterWrite.SUBMV_ParamTimeOutConnect) , VarOut := ADR(A1_SUBMV.ParamTimeOutConnect), Size:=SIZEOF(A1_SUBMV.ParamTimeOutConnect) ); 
FB_WriteOnChange[80](VarInput := ADR(AllDataParameterWrite.SUBMV_ParamTimeOutDisconnect) , VarOut := ADR(A1_SUBMV.ParamTimeOutDisconnect), Size:=SIZEOF(A1_SUBMV.ParamTimeOutDisconnect) ); 
FB_WriteOnChange[81](VarInput := ADR(AllDataParameterWrite.SUBMV_ParamTempoComAlarm) , VarOut := ADR(A1_SUBMV.ParamTempoComAlarm), Size:=SIZEOF(A1_SUBMV.ParamTempoComAlarm) ); 
FB_WriteOnChange[82](VarInput := ADR(AllDataParameterWrite.SUBMV_ParamPmax) , VarOut := ADR(A1_SUBMV.ParamPmax), Size:=SIZEOF(A1_SUBMV.ParamPmax) ); 
FB_WriteOnChange[83](VarInput := ADR(AllDataParameterWrite.SUBMV_ParamPmin) , VarOut := ADR(A1_SUBMV.ParamPmin), Size:=SIZEOF(A1_SUBMV.ParamPmin) ); 
FB_WriteOnChange[84](VarInput := ADR(AllDataParameterWrite.WS_ParamDurationIntegerGTI) , VarOut := ADR(A1_WS.ParamDurationIntegerGTI), Size:=SIZEOF(A1_WS.ParamDurationIntegerGTI) ); 
*)
END_METHOD

METHOD M_Wago
VAR_INPUT
END_VAR
(*
OpcUaServer_1:=  OpcUa.AllDataR.PP.MesU ; 
OpcUaServer_2:=  OpcUa.AllDataR.PP.MesFreq ; 
OpcUaServer_3:=  OpcUa.AllDataR.PP.OUT_SetptP ; 
OpcUaServer_4:=  OpcUa.AllDataR.PP.OUT_SetptQ ; 
OpcUaServer_5:=  OpcUa.AllDataR.PTR[1].MesDataExd.MesData.MesP ; 
OpcUaServer_6:=  OpcUa.AllDataR.PTR[1].MesDataExd.MesData.MesQ ; 
OpcUaServer_7:=  OpcUa.AllDataR.PTR[1].MesDataExd.MesData.MesI ; 
OpcUaServer_8:=  OpcUa.AllDataR.SUBMV.MesDataExd.MesData.MesU ; 
OpcUaServer_9:=  OpcUa.AllDataR.SUBMV.MesDataExd.MesData.MesFreq ; 
OpcUaServer_10:=  OpcUa.AllDataR.WS.MesGTI ; 
OpcUaServer_11:=  OpcUa.AllDataR.WS.MesGHI ; 
OpcUaServer_12:=  OpcUa.AllDataR.PTR[1].AX_INV[1].MesDataExd.MesData.MesP ; 
OpcUaServer_13:=  OpcUa.AllDataR.PTR[1].AX_INV[1].MesDataExd.MesData.MesQ ; 
OpcUaServer_14:=  OpcUa.AllDataR.PTR[1].AX_INV[1].MesDataExd.MesData.MesPdc ; 
OpcUaServer_15:=  OpcUa.AllDataR.PTR[1].AX_INV[1].MesDataExd.MesData.MesUdc ; 
OpcUaServer_16:=  OpcUa.AllDataR.PTR[1].AX_INV[1].MesDataExd.MesData.MesU ; 
OpcUaServer_17:=  OpcUa.AllDataR.PTR[1].AX_INV[1].MesDataExd.MesData.MesI ; 
OpcUaServer_18:=  OpcUa.AllDataR.PTR[1].AX_INV[1].MesDataExd.MesData.MesFreq ; 
OpcUaServer_19:=  OpcUa.AllDataR.PTR[1].AX_INV[1].MesDataExd.MesData.OUT_SetptP ; 
OpcUaServer_20:=  OpcUa.AllDataR.PTR[1].AX_INV[1].MesDataExd.MesData.OUT_SetptQ ; 
OpcUaServer_21:=  OpcUa.AllDataR.SUBMV.GRID.MesDataExd.MesData.OUT_SetptP ; 
OpcUaServer_22:=  OpcUa.AllDataR.SUBMV.GRID.MesDataExd.MesData.OUT_SetptQ ; 
OpcUaServer_23:=  OpcUa.AllDataR.SUBMV.ProtectRelay_Freq.MesI  ; 
OpcUaServer_24:=  OpcUa.AllDataR.SUBMV.ProtectRelay_Freq.MesFreq ; 
OpcUaServer_25:=  OpcUa.AllDataR.SUBMV.PM.MesFreq ; 
OpcUaServer_26:=  OpcUa.AllDataR.SUBMV.PM.MesP ; 
OpcUaServer_27:=  OpcUa.AllDataR.SUBMV.PM.MesQ ; 
OpcUaServer_28:=  OpcUa.AllDataR.SUBMV.PM.MesI ; 
OpcUaServer_29:=  OpcUa.AllDataR.SUBMV.PM.MesU ; 
OpcUaServer_30:=  OpcUa.AllDataR.SUBMV.ProtectRelay_Freq.MesI ; 
OpcUaServer_31:=  OpcUa.AllDataR.SUBMV.ProtectRelay_Freq.MesFreq ; 
OpcUaServer_32:=  OpcUa.AllDataR.WS.Pyran_GHI_1.Value ; 
OpcUaServer_33:=  OpcUa.AllDataR.WS.Pyran_GHI_2.Value ; 
OpcUaServer_34:=  OpcUa.AllDataR.WS.Pyran_GTI_1.Value ; 
OpcUaServer_35:=  OpcUa.AllDataR.WS.Pyran_GTI_2.Value ; 
OpcUaServer_36:=  OpcUa.AllDataR.WS.TempSensor_Ext.Value ; 
OpcUaServer_37:=  OpcUa.AllDataR.WS.windDir.Value ; 
OpcUaServer_38:=  OpcUa.AllDataR.WS.WindSp.Value ; 
OpcUaServer_39:=  OpcUa.AllDataR.WS.Rain.AvgmmHour ; 
OpcUaServer_40:=  OpcUa.AllDataR.WS.Rain.AvgmmDay ; 
OpcUaServer_41:=  OpcUa.AllDataR.WS.Rain.AvgmmMonth ; 
OpcUaServer_42:=  OpcUa.AllDataR.WS.TempSensor_Panel_PTR1.Value ; 
OpcUaServer_43:=  OpcUa.AllDataR.WS.TempSensor_Panel_PTR2.Value ; 
*)
END_METHOD

END_PROGRAM

// ---- 00_FunctionsBlocks/Beckhoff/AlarmManagement/SMS_Server.TcPOU
PROGRAM SMS_Server
VAR PERSISTENT
	AX_Numtel						: ARRAY[1..CstNbUser] OF STRING(26) ;	//Contient tous les numéros des utilisateurs
	AX_Subscribed					: ARRAY[1..CstNbUser] OF BOOL ;			//Contient tous les états d'abonnements des utilisateurs aux SMS
	AX_NomUtili						: ARRAY[1..CstNbUser] OF STRING(50);	//Contient tous les noms des utilisateurs
	AX_User_LVL						: ARRAY[1..CstNbUser] OF WORD;			//Contient tous les niveau d'adhésion des utilisateurs.
END_VAR

VAR_INPUT
	IN_DataSetFifo_ReadSMS			: FB_SMSDatasetFifo_Read; //Buffer automate des sms récuperer depuis modem Gsm
	IN_DataSetFifo_SendSMS			: FB_SMSDatasetFifo_Send; //Buffer automate des sms récuperer depuis modem Gsm	
	IN_AX_Journal					: ARRAY [0..CstNbAlarmCode] OF ARRAY[0..15] OF ST_ValuesAlarms; //Journal d'envoi, contient destinataire et message, et gestion de l'envois ou pas du sms
	IN_Reset_OPC					: BOOL;
	IN_ChangePhoneMailInfos_OPC			: BOOL;
	IN_Reset_SmsServer				: BOOL;
	IN_CmdReset_L					: BOOL;
	IN_CmdDeleteAllSms			: BOOL;
END_VAR

VAR
	fbSerialLineControl		: SerialLineControl;
	stTxBufferPC			: ComBuffer;
	stRxBufferPC			: ComBuffer;
	fbReadSMS				: FB_ReadSMS;
	fbSendSMS				: FB_SendSMS;
	fbDeleteSMS				: FB_DeleteSMS;
	fbDeleteAllSMS			: FB_DeleteAllSMS;
	Fblogin 				: FB_Login;
	
	//READ VARIABLE 
	bStartRead				: BOOL; //Gestion du front montant FB ReadSMS
	ReadSMS_bBusy			: BOOL;
	ReadSMS_bError			: BOOL;
	ReadSMS_nErrorID		: UINT;
	
	LoginSMS_bError			: BOOL;
	LoginSMS_bBusy		    : BOOL;
	IndexReadMessage		: USINT:=1; //Index du message a lire
	ReadSMS_MessageText		: STRING(240); // Message brut du SMS recu
	Etape_Read 		 		: SINT:=0; // Etape du Case de M_Fill_Buffer_Read
	Message_Tous_lu 		: BOOL;  // Si tous les message du buffer READ sont lu : True sinon False
	
	//DELETE VARIABLE
	bStartDelete			: BOOL; //Gestion du front montant FB DeleteSms
	DeletedSMS_bBusy		: BOOL;
	DeletedSMS_Error		: BOOL;
	DeletedSMS_nErrorID		: UINT;
	
	IndexDeleteMessage 		: USINT:=1; //Index du message a supprimer
	
	//SEND VARIABLE
	bStartSend				: BOOL;
	Message_Send			: STRING(160);
	MesTimeStamp			: STRING(17);
	SendSMS_bBusy			: BOOL;
	SendSMS_bError			: BOOL;
	Etape_Send				: SINT;
	CPT						: SINT:=1;
	Num_Tel					: STRING(30);

	//INIT VARIABLE
	bStartlogin             : BOOL:=TRUE; //Gestion du front montant FB login
	bInit					: BOOL;
	
	//Variables de All Delete
	DeletedAllSMS_bBusy		: BOOL;
	DeletedAllSMS_Error		: BOOL;
	DeletedAllSMS_nErrorID	: UINT;
	G7_DelAll				: SINT;

	Bstart_delete_all		: BOOL;    
	
	//M_G7_SMS
	CPT_Message				: CTU;
	


	//TABLEAU
	AX_MesAlarmCode_Bool	: ARRAY [1..CstNbAlarmCode] OF ARRAY[1..15] OF BOOL; //Tableau de tous les alarmesCode en Bool
	AX_Alarm_State			: ARRAY [1..CstNbAlarmCode] OF ARRAY[1..15] OF BOOL; //Tableau de Bool avec toutes les nouveaux bit modifiés
	fbXorWord				: FB_XorWord; //Compare 2 Word et retourne les bit modifié
	Extract_Num_Mes			: FB_Extract_Num_Mes; //Extraction des infos: Message,Numero de tel

	// M_Evaluate
	MesData			: ServerSMS;
	CalNbrUtiliActive    : INT := 10;
	//AlarmCode
	RS_LoginSMS_bError		: RS;
	RS_SendSMS_bError       : RS;
	RS_ReadSMS_bError       : RS;
	RS_DeletedSMS_Error     : RS;
    RS_DeletedAllSMS_Error  : RS;

	AX_Cmd_SMS				: ARRAY[1..CstNbCMD] OF STRING(26):=['Infos','Reboot_ADSL','P_Onduleur','Stop_SMS','Start_SMS','Toggle subscription','Ip Publique','Active Alarms','Help','Test SMS','ForcedStayConnect','Restart HHCollector','Restart PLC','Auto Couplage','Disconnect', 'VPN Connect', 'VPN Disconnect', 'Reboot_IPC']; //Contient toutes les commandes possibles

	Serial_Use				: BOOL:=TRUE;
	ReadAct					: BOOL:=FALSE;
	LoginOK                 : BOOL:=TRUE;
	Reset					: BOOL;
	
	//OPC
	RS_OPC					: RS;
	RS_Deletteall			: RS;
	RS_Reset				: RS;
	Trig_OPC				: R_TRIG;
	Trig_OpcDelAll			: R_TRIG;
	Trig_OpcReset			: R_TRIG;

	
	
END_VAR

IF NOT bInit THEN
	M_Init();
ELSE
	
	// READ OPC Data .
	M_OPC();

	//SERIALLINEMODE_EL6_22B	
	fbSerialLineControl(Mode:= SERIALLINEMODE_PC_COM_PORT ,
		pComIn:= ADR(stPCComInData),
		pComOut:= ADR(stPCComOutData),
		SizeComIn:= UINT_TO_INT( SIZEOF(stPCComInData)),
		TxBuffer:= stTxBufferPC,
		RxBuffer:= stRxBufferPC,
		Error=> ,
		ErrorID=> );
		
	Fblogin(bStart:=bStartlogin ,					// etrangement le login fonctionne puis fait une erreur , puis refonctionne etc . relance du login sur read error je pense qui entraine une tentative de login qui foire. 	
			stTxBuffer:=stTxBufferPC,	
			stRxBuffer:=stRxBufferPC,
			bBusy =>LoginSMS_bBusy,
			bError=>LoginSMS_bError
			);		
		
	fbSendSMS(bStart:= bStartSend,
		sPhoneNumber:= Num_Tel,
		bReset := IN_Reset_OPC ,
		sSMSText:= Message_Send,
		stTxBuffer:=stTxBufferPC ,
		stRxBuffer:=stRxBufferPC,
		bBusy=>SendSMS_bBusy,
		bError=>SendSMS_bError);
	
	fbReadSMS(bStart:= bStartRead,
		nIndex:= IndexReadMessage,
		stTxBuffer:=stTxBufferPC ,
		stRxBuffer:=stRxBufferPC ,
		bBusy=> ReadSMS_bBusy,
		bError=> ReadSMS_bError,
		nErrorID=> ReadSMS_nErrorID
		);
	
	
	fbDeleteSMS
	(
		bStart:= bStartDelete,
		nIndex:= IndexDeleteMessage,
		stTxBuffer:=stTxBufferPC,
		stRxBuffer:=stRxBufferPC,
		bBusy=> DeletedSMS_bBusy,
		bError=> DeletedSMS_Error,
		nErrorID=> DeletedSMS_nErrorID
	);
	
	fbDeleteAllSMS
	(
		bStart:= Bstart_delete_all,
		stTxBuffer:=stTxBufferPC,
		stRxBuffer:=stRxBufferPC,
		bBusy=> DeletedAllSMS_bBusy,
		bError=> DeletedAllSMS_Error,
		nErrorID=> DeletedAllSMS_nErrorID
	);	

	M_DeleteAll();
	M_Fill_Buffer_Read(); //Lecture de tous les messages recu

	M_AlarmManager();
	M_Evaluate();		// Update serveur info
	M_Send(); // Envois de tous les messages (Alarm ou réponce aux sms de cmd)

	M_Cmd_Execute(); // Verification des messages recu
	
	IF Reset OR IN_Reset_OPC  THEN
		M_Reset();
	END_IF
	
	IF NOT LoginSMS_bBusy AND NOT LoginSMS_bError AND LoginOK THEN
		BstartLogin := FALSE;
		Serial_Use:=FALSE;
		LoginOK:=FALSE;
	END_IF
	
	
END_IF

METHOD M_AlarmManager
VAR
	ii:SINT;
	jj:INT;
	KK:INT;
	FB_AlarmCodeManager			: FB_AlarmCodeManager ;
END_VAR
RS_LoginSMS_bError(SET:=LoginSMS_bError,RESET1:=	IN_CmdReset_L OR IN_Reset_OPC); 		
RS_SendSMS_bError(SET:=SendSMS_bError,RESET1:=  	IN_CmdReset_L OR IN_Reset_OPC); 		
RS_ReadSMS_bError(SET:=ReadSMS_bError,RESET1:=  	IN_CmdReset_L OR IN_Reset_OPC); 		
RS_DeletedSMS_Error(SET:=DeletedSMS_Error,RESET1:=	IN_CmdReset_L OR IN_Reset_OPC); 		
RS_DeletedAllSMS_Error(SET:=DeletedAllSMS_Error,RESET1:=IN_CmdReset_L OR IN_Reset_OPC); 	

// ALARM CODE //
	FB_AlarmCodeManager(
		bAlarm1			:= RS_LoginSMS_bErrOR.Q1		  ,			// Login SMS Error
		bAlarm2			:= RS_SendSMS_bErrOR.Q1		   ,			// Send SMS Error
		bAlarm3			:= RS_ReadSMS_bErrOR.Q1		   ,			// Read SMS Error 
		bAlarm4			:= RS_DeletedSMS_ErrOR.Q1		 ,			// Delete SMS Error 
		bAlarm5			:= RS_DeletedAllSMS_ErrOR.Q1	,			// Delete All Sms Error
		bAlarm6			:= IN_DataSetFifo_ReadSMS.bOverwrite,		// Read Fifo overflow
		bAlarm7			:= IN_DataSetFifo_SendSMS.bOverwrite,       // Send Fifo overflow
		bAlarm8			:= FALSE,                                   //
		bAlarm9			:= FALSE,                                   //
		bAlarm10		:= FALSE,                                   //
		bAlarm11		:= FALSE,									//
		bAlarm12		:= FALSE,                                   //
		bAlarm13		:= FALSE,                                   //
		bAlarm14		:= FALSE,                                   //
		bAlarm15		:= FALSE,                                   //
		wAlarmCode		=>MesData.MesAlarmCode);
END_METHOD

METHOD M_Cmd_Execute
VAR_INPUT
END_VAR

VAR
	i: SINT;
	Num_Valide 		: BOOL;
	Message_Valide 	: BOOL;
	Index_CMD 		: SINT;
END_VAR
IF IN_DataSetFifo_ReadSMS.nCount > 0 THEN
	IN_DataSetFifo_ReadSMS.A_Get(); // Récuperation du FIFO
	FOR i:=1 TO CstNbUser DO // VERIFICATION du numéro de telephone
		IF AX_Numtel[i]=IN_DataSetFifo_ReadSMS.Out.Num THEN
			Num_Valide := TRUE;
			EXIT;
		END_IF
	END_FOR
	IF Num_Valide THEN
		FOR i:=1 TO CstNbCMD DO // VERIFICATION du message
			IF IN_DataSetFifo_ReadSMS.Out.Message=AX_Cmd_SMS[i] THEN
				Message_Valide := TRUE;
				Index_CMD:=i;
				EXIT;
			END_IF
		END_FOR
	END_IF
	
	IF Num_Valide AND Message_Valide THEN
		M_G7_SMS(G7_Etape:=Index_CMD);

	ELSE
		IN_DataSetFifo_ReadSMS.A_Remove(); //IL s'agit d'un spam ou d'un utilisateur non autorisé
	END_IF
	

END_IF
END_METHOD

METHOD M_DeleteAll


VAR
	
END_VAR
CASE G7_DelAll OF
	
	0: // Entrée
		IF RS_Deletteall.Q1 AND NOT Serial_Use THEN
			Serial_Use 			:= TRUE;
			Bstart_delete_all 	:= TRUE;
			G7_DelAll 			:= 1;
		END_IF
	1: // attente du bb=usy
		Bstart_delete_all 	:= FALSE;
		IF NOT DeletedAllSMS_bBusy OR DeletedAllSMS_Error THEN
			RS_Deletteall(RESET1:= TRUE);
			RS_Deletteall(RESET1:= FALSE);
			Serial_Use 			:= FALSE;
			G7_DelAll 			:= 0;
		END_IF
		
		
END_CASE
END_METHOD

METHOD M_Evaluate
VAR 
	KK: INT;
END_VAR
CalNbrUtiliActive := 0 ;
FOR KK:=1 TO CstNbUser DO 
	IF 	AX_Numtel[KK] <> '' THEN 
		CalNbrUtiliActive := CalNbrUtiliActive+1 ; 
	END_IF
END_FOR



Mesdata.NbrUtiliActive 	:= CalNbrUtiliActive ;
Mesdata.AX_Numtel		:= AX_Numtel			;
Mesdata.AX_Subscribed	:= AX_subscribed	    ;
MesData.AX_NomUtili		:= AX_NomUtili		    ;
MesData.AX_UserLVL		:= AX_User_LVL		    ;
END_METHOD

METHOD M_Fill_Buffer_Read
CASE Etape_Read OF
	0://Initilisation
		IF NOT ReadSMS_bBusy AND NOT Serial_Use AND ReadAct THEN
			Etape_Read:=10;
			ReadSMS_MessageText:='';
			bStartlogin:=TRUE;
			Serial_Use:=TRUE;
		END_IF
	10: //Initialisation MODEM (ECHO OFF)
		//Serial_Use:=TRUE;
		bStartlogin:=FALSE;
		IF NOT LoginSMS_bBusy AND NOT LoginSMS_bError THEN
			Etape_Read:=1;
			BstartRead:=TRUE;	
		ELSIF LoginSMS_bError THEN
			Etape_Read:=0;
			Serial_Use:=FALSE;
		END_IF
	1://Lecture des sms
		//GVL_Rapale.Serial_Use:=TRUE;
		ReadSMS_MessageText:=fbReadSMS.sMessageText;
		BstartRead:=FALSE;	
		IF NOT ReadSMS_bBusy AND NOT ReadSMS_bError THEN	
			Etape_Read:=2;
			Serial_Use:=FALSE;
		ELSIF ReadSMS_bError THEN
			Etape_Read:=0;
			Serial_Use:=FALSE;
			
		END_IF
		
	2://Analyse du sms en Cas d'un message non vide
		IF(ReadSMS_MessageText<>'OK$R$N') AND (ReadSMS_MessageText<>'') THEN
			
			IF (FIND(ReadSMS_MessageText,'REC UNREAD')>0) THEN		//
				Message_Tous_lu := FALSE;
				IndexReadMessage:=IndexReadMessage+1;
				Extract_Num_Mes(InMessage:=ReadSMS_MessageText);
				IN_DataSetFifo_ReadSMS.A_Add( in := Extract_Num_Mes.OutDataEntry);
				Etape_Read:=0;					
			ELSE	// Messages have already been read. 
				Message_Tous_lu := TRUE;
				IndexReadMessage:=IndexReadMessage+1;
				ReadSMS_MessageText:='';
				Etape_Read:=0;
			END_IF
		ELSE
			Etape_Read:=3;
		END_IF
	3://Analyse du sms en cas de message vide
		IF Message_Tous_lu THEN
			Etape_Read:=4;
		ELSE
			IndexReadMessage:=1;
			Etape_Read:=0;
		END_IF
	4://Initialisation du Delete_FB
		IF NOT DeletedSMS_bBusy AND ReadAct THEN //AND NOT GVL_Rapale.Serial_Use THEN
			Etape_Read:=5;
			bStartDelete:=TRUE;
			Serial_Use:=TRUE;
		END_IF
	5://Suppression du buffer GSM
		//GVL_Rapale.Serial_Use:=TRUE;
			bStartDelete:=FALSE;
		IF NOT DeletedSMS_bBusy AND NOT DeletedSMS_Error THEN
			Serial_Use:=FALSE;
			Etape_Read:=6;
		ELSIF DeletedSMS_Error THEN
			//GVL_Rapale.Serial_Use:=FALSE;
			Etape_Read:=4;
			Serial_Use:=FALSE;
		END_IF
	6://Controle suppression
		IF IndexDeleteMessage=IndexReadMessage-1 THEN
			Etape_Read:=0;
			IndexDeleteMessage:=1;
			Message_Tous_lu:=FALSE;
			IndexReadMessage:=IndexReadMessage+1;
			Serial_Use:=FALSE;
		ELSE
			IndexDeleteMessage:=IndexDeleteMessage+1;
			Etape_Read:=4;
		END_IF		
		
END_CASE
END_METHOD

METHOD M_G7_SMS
VAR_INPUT
	G7_Etape :SINT;
END_VAR

VAR
	InStruct 		: ST_ValuesAlarms;
END_VAR
FUN_Alarms.M_G7_SMS(
	DataSetFifo_ReadSMS		:= IN_DataSetFifo_ReadSMS,
    IN_DataSetFifo_SendSMS	:= IN_DataSetFifo_SendSMS,
 	CPT_Message				:= CPT_Message,	
    InStruct 				:= InStruct,
    G7_Etape 				:= G7_Etape,
    AX_Numtel				:= AX_Numtel,
    AX_subscribed			:= AX_subscribed,
    AX_MesAlarmCode_Bool	:= AX_MesAlarmCode_Bool,
    AX_Cmd_SMS		        := AX_Cmd_SMS
);
END_METHOD

METHOD M_Init

//Initialisation BUFFER

	//Buffer pour la lecture des sms
	IN_DataSetFifo_ReadSMS.A_Reset();
	IN_DataSetFifo_ReadSMS.A_Add();
	IN_DataSetFifo_ReadSMS.A_Get();
	IN_DataSetFifo_ReadSMS.A_Remove();
	
	//Buffer pour l'envois des sms
	IN_DataSetFifo_SendSMS.A_Reset();
	IN_DataSetFifo_SendSMS.A_Add();
	IN_DataSetFifo_SendSMS.A_Get();
	IN_DataSetFifo_SendSMS.A_Remove();

//Initialisation du Journal		
bInit := TRUE;
END_METHOD

METHOD M_OPC : BOOL
VAR
	AX_Numtel_Init				: ARRAY[1..CstNbUser] OF STRING(26);
END_VAR
Trig_OPC(CLK := IN_ChangePhoneMailInfos_OPC);
Trig_OpcDelAll(CLK := IN_CmdDeleteAllSms);
Trig_OpcReset(CLK:= IN_Reset_SmsServer);

RS_OPC(SET:= Trig_OPC.Q);
RS_Deletteall(SET:=Trig_OpcDelAll.Q);
RS_Reset(Set:=Trig_OpcReset.Q);

IF (*NOT Serial_Use AND*) RS_OPC.Q1 THEN
	//Numéro de téléphone
	AX_Numtel := OpcUa.AllValueW.AX_NbPhone_OPC;
	//Nom d'utilisateur
	AX_NomUtili	:= OpcUa.AllValueW.AX_NamesUsers_OPC;
	
	// User LVL . 
	AX_User_LVL := OpcUa.AllValueW.AX_UserLVL;

	//Gestion subscription
	AX_Subscribed := OpcUa.AllValueW.AX_SubscribedSms_OPC;

	RS_OPC(RESET1:= TRUE);
	RS_OPC(Reset1 := FALSE);
END_IF

IF RS_Reset.Q1 THEN
	IN_Reset_Opc := TRUE;
END_IF
END_METHOD

METHOD M_Reset : BOOL
VAR_INPUT
END_VAR
IN_DataSetFifo_SendSMS.A_Reset();

bStartRead 		:= FALSE;
bStartSend 		:= FALSE;
bStartDelete 	:= FALSE;
bStartlogin 	:= FALSE;
Serial_Use		:= FALSE;


SendSMS_Berror := FALSE ;
ReadSMS_bError := FALSE ;
LoginSMS_bError := FALSE ; 
DeletedSMS_Error := FALSE ; 
DeletedAllSMS_Error := FALSE ; 

RS_Reset(RESET1 := TRUE);
RS_Reset(RESET1 := FALSE);
Reset 			:= FALSE;
IN_Reset_OPC 		:= FALSE;
END_METHOD

METHOD M_Send
VAR_INPUT
END_VAR

CASE ETAPE_Send OF
	0://Etape d'entree
		IF NOT SendSMS_bBusy  AND NOT Serial_Use AND IN_DataSetFifo_SendSMS.nCount > 0 AND NOT LoginSMS_bBusy AND NOT LoginSMS_bError THEN  //Si serial libre et buffer contient plus d'une infos
			ReadAct:=FALSE;	
			Serial_Use:=TRUE;
			//bStartSend:=TRUE;
			SendSMS_bError := FALSE;
			Num_Tel := '';
			Message_Send:='';
			IN_DataSetFifo_SendSMS.A_Get();  //recuperation du message dans le send buffer 
			ETAPE_Send := 20  ; 
		ELSE
			ReadAct:=TRUE;	// En attente de lecture de mot d'alarme
		END_IF
			
		20:// Check les utilisateurs pour l'envoi des SMS 
			IF AX_Numtel[CPT] <> '' AND  AX_Subscribed[CPT] AND IN_DataSetFifo_SendSMS.out.Num_tel = '' AND (AX_User_LVL[CPT] AND IN_DataSetFifo_SendSMS.out.Alarms_LVL)>0    THEN
				// On envoi l'alarme si l'utilisateur est subscribed , et est dans la liste de diffusion de l'alarme
				Num_Tel:=AX_NumTel[CPT];
				bStartSend:=TRUE;
				ETAPE_Send:=1;
				MesTimeStamp := CONCAT(REPLACE(STR1:= IN_DataSetFifo_SendSMS.Out.TimeStamp_Act, STR2 := ' ', L := 1, P := 11), ' ') ;

				Message_Send := CONCAT(str1:=CONCAT(str1:=CONCAT(str1:=MesTimeStamp, str2:='$NID:' ), STR2:= UINT_TO_STRING(IN_DataSetFifo_SendSMS.out.ID)), STR2:=' ,' ) ; 
				Message_Send := CONCAT(STR1:=Message_Send , STR2:= IN_AX_Journal[IN_DataSetFifo_SendSMS.out.IndexWord][IN_DataSetFifo_SendSMS.Out.IndexBit].Message);
				
				IF IN_DataSetFifo_SendSMS.OUT.Active  THEN //Connaitre le statut de l'alarme: Active ou Non active
					Message_Send:=Concat(left(Message_Send, 125),' : Active');	// ajout de la mention activee ou desactive 
				ELSE
					Message_Send:=concat(left(Message_Send, 125),' : Desactive');
				END_IF
			ELSIF ( NOT AX_Subscribed[CPT] OR (AX_User_LVL[CPT] AND IN_DataSetFifo_SendSMS.out.Alarms_LVL)=0  ) AND IN_DataSetFifo_SendSMS.out.Num_tel = ''  THEN
				// L'alarme n'est pas envoyéeà cet utilisateur	
				Num_Tel := '';
				ETAPE_Send:=2;
			ELSIF IN_DataSetFifo_SendSMS.out.Num_tel <> ''  THEN
				// Si un numero de telephone est renseigné précisement, on envoi à ce numéro quelque soit la liste de diffusion , ou si l'utilisateur est subscribed
				bStartSend:=TRUE;
				Message_Send := CONCAT(STR1:=Message_Send , STR2:= IN_AX_Journal[IN_DataSetFifo_SendSMS.out.IndexWord][IN_DataSetFifo_SendSMS.Out.IndexBit].Message);
				Num_Tel:=IN_DataSetFifo_SendSMS.Out.Num_tel;
				ETAPE_Send:=1;
			ELSE
				// L'alarme n'est pas envoyée		
				Num_Tel := '';
				ETAPE_Send:=2;
			END_IF

	1://Envois du message
		Bstartsend:=FALSE;	
		IF NOT SendSMS_bBusy  THEN
			IF IN_DataSetFifo_SendSMS.OUT.IndexWord > 0 AND IN_DataSetFifo_SendSMS.In.Num_tel = ''   THEN
				ETAPE_Send:=2; // Alarme
				
			ELSE
				ETAPE_Send:=3; // Retour Sms ou utilisateur de renseignée
			END_IF
		ELSIF NOT SendSMS_bBusy AND SendSMS_Berror THEN // GGY
			//ETAPE_Send:=0; modif lWN seminaire 26/08/2020, gestion des ATE0, si erreur on supprime tout de meme le sms.
			ETAPE_Send:= 3;
			SendSMS_Berror := FALSE ; // On reset l'error apres avoir supprimé le SMS . 
			
		END_IF
		
	2:// Switch a un autre utilisateur
		IF CPT< CstNbUser THEN
			CPT:=CPT+1;
			ETAPE_Send:=20;
		ELSE
			ETAPE_Send:=3;
		END_IF
	
	3://Suppression de l'alarme et on passe au prochaine element dans le fifo
		IN_DataSetFifo_SendSMS.A_Remove();
		CPT:=1;
		Message_Send:='';
		ETAPE_Send:=0;
		Serial_Use:=FALSE;
		bStartSend:=FALSE;

END_CASE
END_METHOD

END_PROGRAM

// ---- 04_Application/MAIN/TEST.TcPOU
PROGRAM TEST
VAR
// create an instance for all FB in base project in order to test if there are errors in the FB ()

	moyenne_test : MOYENNE;
	time_Test : TIME := T#5s;
	bTest : BOOL;
	rValue : REAL;
	
END_VAR


moyenne_test(
	In_fenetre_mesure := time_Test,
	In_synchro := CalLocalTimeStruct.wSecond MOD 5 = 0,
	In_valeur := word_to_real(CalLocalTimeStruct.wSecond)
);
moyenne_test.Calcul();

END_PROGRAM

// ---- 04_Application/ALARM/FUN_Alarms.TcPOU
PROGRAM FUN_Alarms
VAR_INPUT
	IN_Directory					: STRING := 'C:\Users\Administrator\Documents\Historisation\';	// Directory where the alarms are saved in csv
	ParamDisableSMS					: BOOL ;	// True : SMS Serveur is disabled 
	AX_MesAlarmCode				: ARRAY [0..CstNbAlarmCode] OF WORD;    // Tableau de Word avec tous les AlarmCode 

END_VAR

VAR_INPUT PERSISTENT
	AX_Journal						: ARRAY [0..CstNbAlarmCode] OF ARRAY[0..15] OF ST_ValuesAlarms; //Journal d'envoi, contient destinataire et message, et gestion de l'envois ou pas du sms
	bFactoryReset					: BOOL:= TRUE ;
END_VAR



VAR
	AX_RecupWord 					: ARRAY [0..CstNbAlarmCode] OF WORD;

	
	// M_ALARMPROCESSING	



		
	//	FB_Flicker					: ARRAY [0..CstNbAlarmCode] OF ARRAY[0..15] OF FB_DetectFlicker ; 
		
	// CSV

	
	//MAIL
		Directory					: STRING;
	//SMS
	
	
	
END_VAR

IF bFactoryReset THEN
	M_Init();
	///////// 
END_IF

M_AlarmManager();
M_AlarmProcessing();
	
// Ici, on prend surtout en compte les alarmes 
FUN_Alarms_CSV(ParamSeparateur := ';',ParamExtension := '.csv');

IF MAIN.OUT_CalRunningPLC_IO THEN
	Directory := SEL(CstPLCBackup , 'C:\TwinCAT\Functions\Annex_Fonctions\SendEmail\' , 'C:\TwinCAT\Functions\Annex_Fonctions\SendEmail_Slave\') ; 
	FUN_SendMail(IN_Directory := Directory , ParamNetID := CstNetAmsId_IndusPC);
	SMS_Server (IN_AX_Journal := AX_Journal);
	InfluxDb_AlarmsManagement() ; 
	//Firebird_WriteAlarms(ParamTimeBetweenReconnect:= T#1M);
END_IF

METHOD M_AlarmManager : BOOL
VAR_INPUT
END_VAR

VAR
	KK : UINT;
	
END_VAR
END_METHOD

METHOD M_AlarmProcessing : BOOL
////////////////// 
// Process alarms, detect changes and segregate if the alarm has to be logged in csv, send by mail, or send by sms
//////////////////


VAR
	LL : UINT;
	KK : UINT;
	
	MesXorWord 		: WORD;
	MesAlarmWord	: WORD;


	IN_AlarmInflux : ST_InfluxAlarmsInsert;
	MesRolAlarmWord: WORD;
	MesRolXoRWord: WORD;
END_VAR
//Retrieve all Alarms word and detect if a change occured. 
FOR KK := 1 TO CstNbAlarmCode DO
	MesXorWord := AX_MesAlarmCode[KK] XOR AX_RecupWord[KK];
	IF MesXorWord > 0 THEN  // Compare si il y a eu des changements dans les alarmes word
		FOR LL := 0 TO 15 DO 
			MesRolXoRWord 	:= ROR(MesXorWord, LL);
			MesRolAlarmWord := ROR(AX_RecupWord[KK], LL);
			
			IF MesRolXoRWord.0 THEN  // Si il y a eu un changement sur le bit
				AX_Journal[KK][LL].Value := MesRolAlarmWord.0; // 
				AX_Journal[KK][LL].TimeStamp_Act:= SYSTEMTIME_TO_STRING(CalLocalTimeStruct);	// On ecrit l'heure du changement
	
				IF (AX_Journal[KK][LL].Value AND AX_Journal[KK][LL].Groupe > 0) OR ( NOT(AX_Journal[KK][LL].Value) AND  AX_Journal[KK][LL].Groupe = 2)  THEN// Il s'agit d'une alarme qu'on doit écrire sur activation

					// CSV alarms :  on ecrit l'alarme
					FUN_Alarms_CSV.FIFO.In := AX_Journal[KK][LL];
					FUN_Alarms_CSV.FIFO.A_Add();
					
					//MAIl alarms
					IF AX_Journal[KK][LL].Alarms_LVL.3 THEN
						FUN_SendMail.FIFO.In := AX_Journal[KK][LL];
						FUN_SendMail.FIFO.A_Add();
					END_IF
					
					InfluxDb_AlarmsManagement.IN_FIFO.In :=  AX_Journal[KK][LL];
					InfluxDb_AlarmsManagement.IN_FIFO.A_Add();
					
					// SMS Alarms. On ecrit si Serveur SMS n'est pas descativé
					IF NOT ParamDisableSMS  AND AX_Journal[KK][LL].Alarms_LVL.4 THEN 
						SMS_Server.IN_DataSetFifo_SendSMS.In.IndexWord		:= KK;
						SMS_Server.IN_DataSetFifo_SendSMS.IN.IndexBit		:= LL;
						SMS_Server.IN_DataSetFifo_SendSMS.IN.Num_tel 		:= '';
						SMS_Server.IN_DataSetFifo_SendSMS.In.ID				:= AX_Journal[KK][LL].ID;
						SMS_Server.IN_DataSetFifo_SendSMS.In.TimeStamp_Act	:= AX_Journal[KK][LL].TimeStamp_Act;						
						SMS_Server.IN_DataSetFifo_SendSMS.IN.Active			:= AX_Journal[KK][LL].Value;	// TRUE si activation. 
						SMS_Server.IN_DataSetFifo_SendSMS.IN.Alarms_LVL		:= AX_Journal[KK][LL].Alarms_LVL ;
						SMS_Server.IN_DataSetFifo_SendSMS.A_Add();
					END_IF 
				END_IF
			END_IF
		END_FOR
		memcpy(destAddr := ADR(AX_MesAlarmCode[KK]), srcAddr :=ADR(AX_RecupWord[KK]), n := SIZEOF(AX_RecupWord[KK])); //On écrase la valeur par la dernière valeur.	
	END_IF
END_FOR
END_METHOD

METHOD M_G7_SMS : BOOL
VAR_IN_OUT
	DataSetFifo_ReadSMS		: FB_SMSDatasetFifo_Read;	
    IN_DataSetFifo_SendSMS		: FB_SMSDatasetFifo_Send;
	CPT_Message				: CTU;
	InStruct 				: ST_ValuesAlarms;
	G7_Etape 				: SINT;
	AX_Numtel				: ARRAY[1..CstNbUser] OF STRING(26);	//Contient tous les numéros des utilisateurs
	AX_Subscribed			: ARRAY[1..CstNbUser] OF BOOL;			//Contient tous les états d'abonnements des utilisateurs aux SMS
	AX_MesAlarmCode_Bool	: ARRAY [1..CstNbAlarmCode] OF ARRAY[1..15] OF BOOL; //Tableau de tous les alarmesCode en Bool
	AX_Cmd_SMS				: ARRAY[1..CstNbCMD] OF STRING(26);
END_VAR

VAR
	Message : STRING(255);
	SUB_MVcalstate			: BYTE;
	SUB_MVData				: SUBMV;
	KK					: INT;
	MM					: INT;
	LL					: INT;
	JJ					: INT;
	ii					: SINT;
	Id_Num				: INT;
	sState				: STRING;

	Etat    			: STRING(255);
	EtatDp1				: STRING(255);
	EtatMainMVCB				: STRING(255);
	FbFormat			: FB_FormatString;
	RestartGsm			: BOOL;
	
	bLocal				: STRING(255);
END_VAR
CPT_Message(PV:=16,CU:=TRUE,RESET:=CPT_Message.Q);
CPT_Message(CU:=FALSE,RESET:=CPT_Message.Q);
CASE G7_Etape OF
	
	1://Commande INFO

		//IF A1_SUBMV.MesDataExd.MesData.MesState.2 THEN 
		//	Etat := 'Decouple, ';
		//ELSIF A1_SUBMV.MesDataExd.MesData.MesState.1 THEN
		//	Etat := 'Couplee, ';
		//ELSIF A1_SUBMV.MesDataExd.MesData.MesState.0 THEN
		//	Etat := 'Effacee, ';
		//END_IF
        //
		//fbFormat(
		//	sFormat:= 'LHERM: %s ; P:%.1f kW; P_PT1: %.1f kW; P_PT2: %.1f kW; P_PT3: %.1f kW; P_PT4: %.1f kW ',
		//	arg1:= F_STRING(Etat), 
		//	arg2:= F_REAL(A1_PP.MesData.MesPsol),  
		//	arg3:= F_REAL(AX_PTR[1].MesDataExd.MesData.MesP), 
		//	arg4:= F_REAL(AX_PTR[2].MesDataExd.MesData.MesP),
		//	arg5:= F_REAL(AX_PTR[3].MesDataExd.MesData.MesP), 
		//	arg6:= F_REAL(AX_PTR[4].MesDataExd.MesData.MesP),
		//	sOut=> Message);
	    //
		//FUN_Alarms.AX_Journal[0][CPT_Message.CV].Message := Message;	
		//IN_DataSetFifo_SendSMS.In.Num_tel:=DataSetFifo_ReadSMS.Out.Num;
		//IN_DataSetFifo_SendSMS.In.IndexWord:=0;
		//IN_DataSetFifo_SendSMS.In.IndexBit:=WORD_TO_SINT(CPT_Message.CV);
		//IN_DataSetFifo_SendSMS.A_Add();
		////DataSetFifo_ReadSMS.A_Remove();
		////2eme message
		//
		//CPT_Message(CU:=TRUE,RESET:=CPT_Message.Q);
		//CPT_Message(CU:=FALSE,RESET:=CPT_Message.Q);
		//fbFormat(
		//	sFormat:= 'Irradiation :PT1GHI: %.1f W/m2; PT1GTI1: %.1f W/m2; PT4GTI_1: %.1f W/m2; PT4GTI_2: %.1f W/m2 ',
		//	arg1:= F_REAl(A1_WS.AX_Pyrano[1].MesData.Value), 
		//	arg2:= F_REAl(A1_WS.AX_Pyrano[2].MesData.Value),   
		//	arg3:= F_REAl(A1_WS.AX_Pyrano[3].MesData.Value), 
		//	arg4:= F_REAl(A1_WS.AX_Pyrano[4].MesData.Value), 
		//	sOut=> Message);
		//	
		//FUN_Alarms.AX_Journal[0][CPT_Message.CV].Message := Message;	
		//IN_DataSetFifo_SendSMS.In.Num_tel:=DataSetFifo_ReadSMS.Out.Num;
		//IN_DataSetFifo_SendSMS.In.IndexWord:=0;
		//IN_DataSetFifo_SendSMS.In.IndexBit:=WORD_TO_SINT(CPT_Message.CV);
		//IN_DataSetFifo_SendSMS.A_Add();
		//
		//////3eme message
		//
		//CPT_Message(CU:=TRUE,RESET:=CPT_Message.Q);
		//CPT_Message(CU:=FALSE,RESET:=CPT_Message.Q);
		//
		//AX_HV_Cel_PDL[1]:= SEL(A1_SUBMV.A1_MainMVCB.MesDataExd.MesData.MesClosed,'Ouvert','Ferme');
		//AX_HV_Cel_PDL[2]:= SEL(A1_SUBMV.AX_FeederMVCB[1].MesDataExd.MesData.MesClosed,'Ouvert','Ferme');
		//AX_HV_Cel_PDL[3]:= SEL(A1_SUBMV.AX_FeederMVCB[1].MesDataExd.MesData.MesClosed,'Ouvert','Ferme');
		//Ax_ETAT_DM1[1]	:= SEL(AX_PTR[1].A1_MainMVCB_PTR.MesDAtaExd.MesData.MesClosed,'Ouvert','Ferme');
		//Ax_ETAT_DM1[2]	:= SEL(AX_PTR[2].A1_MainMVCB_PTR.MesDAtaExd.MesData.MesClosed,'Ouvert','Ferme');
		//Ax_ETAT_DM1[3]	:= SEL(AX_PTR[3].A1_MainMVCB_PTR.MesDAtaExd.MesData.MesClosed,'Ouvert','Ferme');
		//Ax_ETAT_DM1[4]	:= SEL(AX_PTR[4].A1_MainMVCB_PTR.MesDAtaExd.MesData.MesClosed,'Ouvert','Ferme');
		//
		//fbFormat(
		//	sFormat:= 'MainMVCB: %s;  FeederMVCB_1: %s ; FeederMVCB_2: %s; MainMVCB_PTR1: %s;  MainMVCB_PTR2: %s;  MainMVCB_PTR3: %s;  MainMVCB_PTR4: %s  ',
		//	arg1:= F_STRING(AX_HV_Cel_PDL[1]), 
		//	arg2:= F_STRING(AX_HV_Cel_PDL[2]),  
		//	arg3:= F_STRING(AX_HV_Cel_PDL[3]), 
		//	arg4:= F_STRING(Ax_ETAT_DM1[1]), 
		//	arg5:= F_STRING(Ax_ETAT_DM1[2]), 
		//	arg6:= F_STRING(Ax_ETAT_DM1[3]), 
		//	arg7:= F_STRING(Ax_ETAT_DM1[4]), 
		//	sOut=> Message);
	    //
		//FUN_Alarms.AX_Journal[0][CPT_Message.CV].Message := Message;
	    //
		//IN_DataSetFifo_SendSMS.In.Num_tel:=DataSetFifo_ReadSMS.Out.Num;
		//IN_DataSetFifo_SendSMS.In.IndexWord:=0;
		//IN_DataSetFifo_SendSMS.In.IndexBit:=WORD_TO_SINT(CPT_Message.CV);
		//IN_DataSetFifo_SendSMS.A_Add();
		//
		//DataSetFifo_ReadSMS.A_Remove();
		//		
		//InStruct.ID := 975;
		//InStruct.Message :=concat(concat('Le numero de telephone ', IN_DataSetFifo_SendSMS.In.Num_tel), 'a fait une demande Infos par SMS') ;
		//InStruct.TimeStamp_Act := SYSTEMTIME_TO_STRING(CalLocalTimeStruct);
		////FUN_Alarms_CSV.M_AddAction_FIFO(InStruct := InStruct); // Alarme sur activation du code
		//FUN_Alarms_CSV.FIFO.In := InStruct ;
		//FUN_Alarms_CSV.FIFO.A_Add() ;
		
	2://Restart Routeur ADSL
		RestartGsm							:= TRUE;
		OpcUa.AllDataWPulse.CmdReset_Router_ADSL		:= TRUE;
		Message :='Le Routeur Adsl va redemarer';
		FUN_Alarms.AX_Journal[0][CPT_Message.CV].Message := Message;	
		IN_DataSetFifo_SendSMS.In.Num_tel:=DataSetFifo_ReadSMS.Out.Num;
		IN_DataSetFifo_SendSMS.In.IndexWord:=0;
		IN_DataSetFifo_SendSMS.In.IndexBit:=WORD_TO_SINT(CPT_Message.CV);
		IN_DataSetFifo_SendSMS.A_Add();
		DataSetFifo_ReadSMS.A_Remove();
	
		InStruct.ID := 976;
		InStruct.Message := concat(concat('Le numero de telephone ', IN_DataSetFifo_SendSMS.In.Num_tel), 'a Restart le routeur ADSL') ;
		InStruct.TimeStamp_Act := SYSTEMTIME_TO_STRING(CalLocalTimeStruct);
		//FUN_Alarms_CSV.M_AddAction_FIFO(InStruct := InStruct); // Alarme sur activation du code
		FUN_Alarms_CSV.FIFO.In := InStruct ;
		FUN_Alarms_CSV.FIFO.A_Add() ;
		
	3://Puissance des onduleurs
		// 1er message 
		fbFormat(
		sFormat:= 'Onduleur PT1O1: %.1f, PT1O2: %.1f, PT2O1: %.1f, PT2O2: %.1f, PT3O1: %.1f, PT3O2: %.1f, PT4O1: %.1f, PT4O2: %.1f',
		arg1:= F_REAL(Ax_PTR[1].AX_INV[1].MesDataExd.MesData.MesP),
		arg2:= F_REAL(Ax_PTR[1].AX_INV[2].MesDataExd.MesData.MesP),
		arg3:= F_REAL(Ax_PTR[2].AX_INV[1].MesDataExd.MesData.MesP),
		arg4:= F_REAL(Ax_PTR[2].AX_INV[2].MesDataExd.MesData.MesP),
		arg5:= F_REAL(Ax_PTR[3].AX_INV[1].MesDataExd.MesData.MesP),
		arg6:= F_REAL(Ax_PTR[3].AX_INV[2].MesDataExd.MesData.MesP),
		arg7:= F_REAL(Ax_PTR[4].AX_INV[1].MesDataExd.MesData.MesP),
		arg8:= F_REAL(Ax_PTR[4].AX_INV[2].MesDataExd.MesData.MesP),
		sOut=> Message);
		
		FUN_Alarms.AX_Journal[0][CPT_Message.CV].Message := Message;	
		IN_DataSetFifo_SendSMS.In.Num_tel:=DataSetFifo_ReadSMS.Out.Num;
		IN_DataSetFifo_SendSMS.In.IndexWord:=0;
		IN_DataSetFifo_SendSMS.In.IndexBit:= WORD_TO_SINT(CPT_Message.CV);
		IN_DataSetFifo_SendSMS.A_Add();		

		DataSetFifo_ReadSMS.A_Remove();
		
		InStruct.ID := 977;
		InStruct.Message := concat(concat('Le numero de telephone ', IN_DataSetFifo_SendSMS.In.Num_tel), 'a demandé la puissance des onduleurs'); 
		InStruct.TimeStamp_Act := SYSTEMTIME_TO_STRING(CalLocalTimeStruct);
		//FUN_Alarms_CSV.M_AddAction_FIFO(InStruct := InStruct); // Alarme sur activation du code
		FUN_Alarms_CSV.FIFO.In := InStruct ;
		FUN_Alarms_CSV.FIFO.A_Add() ;
		
	4://Mise en pause des alarmes
		ParamDisableSMS := TRUE;
		Message :='Les alarmes SMS sont desactivees';
		FOR MM := 1 TO CstNbUser DO	
			IF AX_Numtel[MM]<>'' THEN
				FUN_Alarms.AX_Journal[0][CPT_Message.CV].Message := Message;	
				IN_DataSetFifo_SendSMS.In.Num_tel:=AX_Numtel[MM];
				IN_DataSetFifo_SendSMS.In.IndexWord:=0;
				IN_DataSetFifo_SendSMS.In.IndexBit:= WORD_TO_SINT(CPT_Message.CV);
				IN_DataSetFifo_SendSMS.A_Add();
				DataSetFifo_ReadSMS.A_Remove();
			END_IF
		END_FOR
		
		InStruct.ID := 978;
		InStruct.Message := concat(concat('Le numero de telephone ', IN_DataSetFifo_SendSMS.In.Num_tel), 'a désactivé les alarmes SMS'); 
		InStruct.TimeStamp_Act := SYSTEMTIME_TO_STRING(CalLocalTimeStruct);
		//FUN_Alarms_CSV.M_AddAction_FIFO(InStruct := InStruct); // Alarme sur activation du code
		FUN_Alarms_CSV.FIFO.In := InStruct ;
		FUN_Alarms_CSV.FIFO.A_Add() ;
	
	5://Start SMS
		ParamDisableSMS := FALSE;
		Message :='Les alarmes SMS sont activees';
		FOR MM := 1 TO CstNbUser DO	
			IF AX_Numtel[MM]<>'' THEN
				FUN_Alarms.AX_Journal[0][CPT_Message.CV].Message := Message;	
				IN_DataSetFifo_SendSMS.In.Num_tel:=AX_Numtel[MM];
				IN_DataSetFifo_SendSMS.In.IndexWord:=0;
				IN_DataSetFifo_SendSMS.In.IndexBit:= WORD_TO_SINT(CPT_Message.CV);
				IN_DataSetFifo_SendSMS.A_Add();
				DataSetFifo_ReadSMS.A_Remove();
			END_IF
		END_FOR
		
		InStruct.ID := 979;
		InStruct.Message := concat(concat('Le numero de telephone ', IN_DataSetFifo_SendSMS.In.Num_tel), 'a réactivé les alarmes SMS'); 
		InStruct.TimeStamp_Act := SYSTEMTIME_TO_STRING(CalLocalTimeStruct);
		//FUN_Alarms_CSV.M_AddAction_FIFO(InStruct := InStruct); // Alarme sur activation du code
		FUN_Alarms_CSV.FIFO.In := InStruct ;
		FUN_Alarms_CSV.FIFO.A_Add() ;
	

 	6:// Unsubscribe
		FOR LL := 1 TO CstNbUser DO
			IF DataSetFifo_ReadSMS.Out.Num = AX_Numtel[LL] THEN
				Id_Num := LL;
				EXIT;
			END_IF
		END_FOR
		AX_Subscribed[Id_Num] := NOT AX_Subscribed[Id_Num];
		sState := SEL(AX_Subscribed[Id_Num], 'Unsubscribed', 'Subscribed');
		Message := Concat('You have toggled your subscription, state =', sState);
		FUN_Alarms.AX_Journal[0][CPT_Message.CV].Message := Message ;
		IN_DataSetFifo_SendSMS.In.Num_tel:=DataSetFifo_ReadSMS.Out.Num;
		IN_DataSetFifo_SendSMS.In.IndexWord:=0;
		IN_DataSetFifo_SendSMS.In.IndexBit:= WORD_TO_SINT(CPT_Message.CV);
		IN_DataSetFifo_SendSMS.A_Add();
		DataSetFifo_ReadSMS.A_Remove();
		
		InStruct.ID := 980;
		InStruct.Message := concat(concat('Le numero de telephone ', IN_DataSetFifo_SendSMS.In.Num_tel), 'a modifie son inscription') ;
		InStruct.TimeStamp_Act := SYSTEMTIME_TO_STRING(CalLocalTimeStruct);
		//FUN_Alarms_CSV.M_AddAction_FIFO(InStruct := InStruct); // Alarme sur activation du code
		FUN_Alarms_CSV.FIFO.In := InStruct ;
		FUN_Alarms_CSV.FIFO.A_Add() ;
		
	7 : 	//Get Public IP 
		fbFormat(
			sFormat:= 'IP publique de la centrale : %s',
			arg1:= F_STRING(ParamIpPublic),
			sOut=> Message);
		
		FUN_Alarms.AX_Journal[0][CPT_Message.CV].Message := Message;	
		IN_DataSetFifo_SendSMS.In.Num_tel:=DataSetFifo_ReadSMS.Out.Num;
		IN_DataSetFifo_SendSMS.In.IndexWord:=0;
		IN_DataSetFifo_SendSMS.In.IndexBit:= WORD_TO_SINT(CPT_Message.CV);
		IN_DataSetFifo_SendSMS.A_Add();
		DataSetFifo_ReadSMS.A_Remove();
		CPT_Message(CU:=TRUE,RESET:=CPT_Message.Q);
		CPT_Message(CU:=FALSE,RESET:=CPT_Message.Q);
		
		InStruct.ID := 981;
		InStruct.Message := concat(concat('Le numero de telephone ', IN_DataSetFifo_SendSMS.In.Num_tel), 'a demandé l IP public ');  
		InStruct.TimeStamp_Act := SYSTEMTIME_TO_STRING(CalLocalTimeStruct);
		//FUN_Alarms_CSV.M_AddAction_FIFO(InStruct := InStruct); // Alarme sur activation du code
		FUN_Alarms_CSV.FIFO.In := InStruct ;
		FUN_Alarms_CSV.FIFO.A_Add() ; 
		
	8: // All Active Alarms
		FOR jj := 1 TO CstNbAlarmCode DO
			FOR ii :=1 TO 15 DO 
				IF(AX_Journal[jj][ii].Value AND (AX_Journal[jj][ii].Alarms_LVL.0 OR AX_Journal[jj][ii].Alarms_LVL.1) AND AX_Journal[jj][ii].Groupe > 0 AND NOT ParamDisableSMS ) THEN // Il s'agit d'une alarme qu'on doit notifier par sms
					IN_DataSetFifo_SendSMS.In.IndexWord	:= jj;
					IN_DataSetFifo_SendSMS.IN.IndexBit		:= ii;
					IN_DataSetFifo_SendSMS.In.Num_tel		:= DataSetFifo_ReadSMS.Out.Num;
					IN_DataSetFifo_SendSMS.IN.Active		:= TRUE;
					IN_DataSetFifo_SendSMS.A_Add();
					CPT_Message(CU:=TRUE,RESET:=CPT_Message.Q);
					CPT_Message(CU:=FALSE,RESET:=CPT_Message.Q);
				END_IF
			END_FOR
		END_FOR
		DataSetFifo_ReadSMS.A_Remove();
		
		InStruct.ID := 982;
		InStruct.Message := concat(concat('Le numero de telephone ', IN_DataSetFifo_SendSMS.In.Num_tel), 'a demandé la liste des alarmes actives');  
		InStruct.TimeStamp_Act := SYSTEMTIME_TO_STRING(CalLocalTimeStruct);
		//FUN_Alarms_CSV.M_AddAction_FIFO(InStruct := InStruct); // Alarme sur activation du code
		FUN_Alarms_CSV.FIFO.In := InStruct ;
		FUN_Alarms_CSV.FIFO.A_Add() ;
		
	9: // Help
		Message :='Les commandes disponibles sont :Infos ';
		FOR KK := 2 TO MIN(7,CstNbCMD) DO // Nbr_CMD-1 DO //pas besoin du Help
			Message := concat(Message, concat('", "',  AX_Cmd_SMS[KK]));
		END_FOR
		FUN_Alarms.AX_Journal[0][CPT_Message.CV].Message := Message;	
		IN_DataSetFifo_SendSMS.In.Num_tel:=DataSetFifo_ReadSMS.Out.Num;
		IN_DataSetFifo_SendSMS.In.IndexWord:=0;
		IN_DataSetFifo_SendSMS.In.IndexBit:=WORD_TO_SINT(CPT_Message.CV);
		IN_DataSetFifo_SendSMS.A_Add();
		
		IF CstNbCMD >7 THEN
			CPT_Message(CU:=TRUE,RESET:=CPT_Message.Q);
			CPT_Message(CU:=FALSE,RESET:=CPT_Message.Q);

			Message :='';
			FOR KK := 8 TO MIN(14,CstNbCMD) DO // Nbr_CMD-1 DO //pas besoin du Help
				Message := concat(Message, concat('", "',  AX_Cmd_SMS[KK]));
			END_FOR	
			FUN_Alarms.AX_Journal[0][CPT_Message.CV].Message := Message;	
			IN_DataSetFifo_SendSMS.In.Num_tel:=DataSetFifo_ReadSMS.Out.Num;
			IN_DataSetFifo_SendSMS.In.IndexWord:=0;
			IN_DataSetFifo_SendSMS.In.IndexBit:=WORD_TO_SINT(CPT_Message.CV);
			IN_DataSetFifo_SendSMS.A_Add();				
		END_IF
		
		IF CstNbCMD >14 THEN
			CPT_Message(CU:=TRUE,RESET:=CPT_Message.Q);
			CPT_Message(CU:=FALSE,RESET:=CPT_Message.Q);

			Message :='';
			FOR KK := 14 TO CstNbCMD DO // Nbr_CMD-1 DO //pas besoin du Help
				Message := concat(Message, concat('", "',  AX_Cmd_SMS[KK]));
			END_FOR	
			FUN_Alarms.AX_Journal[0][CPT_Message.CV].Message := Message;	
			IN_DataSetFifo_SendSMS.In.Num_tel:=DataSetFifo_ReadSMS.Out.Num;
			IN_DataSetFifo_SendSMS.In.IndexWord:=0;
			IN_DataSetFifo_SendSMS.In.IndexBit:=WORD_TO_SINT(CPT_Message.CV);
			IN_DataSetFifo_SendSMS.A_Add();				
		END_IF
		
		DataSetFifo_ReadSMS.A_Remove();
			
		InStruct.ID := 983;
		InStruct.Message := concat(concat('Le numero de telephone ', IN_DataSetFifo_SendSMS.In.Num_tel), 'a demandé la commande Help'); 
		InStruct.TimeStamp_Act := SYSTEMTIME_TO_STRING(CalLocalTimeStruct);
		//FUN_Alarms_CSV.M_AddAction_FIFO(InStruct := InStruct); // Alarme sur activation du code
		FUN_Alarms_CSV.FIFO.In := InStruct ;
		FUN_Alarms_CSV.FIFO.A_Add() ;
	
10: // test d'envois sms
		OPCUA.AllDataWPulse.CmdTestSms := TRUE;
		DataSetFifo_ReadSMS.A_Remove();
		
		InStruct.ID := 984;
		InStruct.Message := concat(concat('Le numero de telephone ', IN_DataSetFifo_SendSMS.In.Num_tel), 'a envoyé une cmd test sms et mail'); 
		InStruct.TimeStamp_Act := SYSTEMTIME_TO_STRING(CalLocalTimeStruct);
		//FUN_Alarms_CSV.M_AddAction_FIFO(InStruct := InStruct); // Alarme sur activation du code
		FUN_Alarms_CSV.FIFO.In := InStruct ;
		FUN_Alarms_CSV.FIFO.A_Add() ;
		
	11: //Forced stay connect Toggle
		A1_PP.ParamForcedStayConnect := NOT A1_PP.ParamForcedStayConnect;
		sState := SEL(A1_PP.ParamForcedStayConnect, 'False', 'True');
		Message := Concat('You have toggled the Variable ForcedStayConnect, state =', sState);
		FUN_Alarms.AX_Journal[0][CPT_Message.CV].Message := Message ;
		IN_DataSetFifo_SendSMS.In.Num_tel:=DataSetFifo_ReadSMS.Out.Num;
		IN_DataSetFifo_SendSMS.In.IndexWord:=0;
		IN_DataSetFifo_SendSMS.In.IndexBit:= WORD_TO_SINT(CPT_Message.CV);
		IN_DataSetFifo_SendSMS.A_Add();
		DataSetFifo_ReadSMS.A_Remove();
		
		InStruct.ID := 985;
		InStruct.Message := concat(concat('Le numero de telephone ', IN_DataSetFifo_SendSMS.In.Num_tel), 'a modifie la variable ForceStauConnect') ;
		InStruct.TimeStamp_Act := SYSTEMTIME_TO_STRING(CalLocalTimeStruct);
		//FUN_Alarms_CSV.M_AddAction_FIFO(InStruct := InStruct); // Alarme sur activation du code
		FUN_Alarms_CSV.FIFO.In := InStruct ;
		FUN_Alarms_CSV.FIFO.A_Add() ;
	
	12: // Restart HH
		OPCUA.AllDataWPulse.CmdRestart_HH := TRUE;
		Message := 'HH collector is restarting';
		FUN_Alarms.AX_Journal[0][CPT_Message.CV].Message := Message ;
		IN_DataSetFifo_SendSMS.In.Num_tel:=DataSetFifo_ReadSMS.Out.Num;
		IN_DataSetFifo_SendSMS.In.IndexWord:=0;
		IN_DataSetFifo_SendSMS.In.IndexBit:= WORD_TO_SINT(CPT_Message.CV);
		IN_DataSetFifo_SendSMS.A_Add();
		DataSetFifo_ReadSMS.A_Remove();
		
		InStruct.ID := 986;
		InStruct.Message := concat(concat('Le numero de telephone ', IN_DataSetFifo_SendSMS.In.Num_tel), 'a redemarre le service HH collecteur') ;
		InStruct.TimeStamp_Act := SYSTEMTIME_TO_STRING(CalLocalTimeStruct);
		//FUN_Alarms_CSV.M_AddAction_FIFO(InStruct := InStruct); // Alarme sur activation du code
		FUN_Alarms_CSV.FIFO.In := InStruct ;
		FUN_Alarms_CSV.FIFO.A_Add() ;
	
	13: // Restart PLC
		OPCUA.AllDataWPulse.CmdRestart_PLC := TRUE;
		Message := 'PLC is restarting Now !';
		FUN_Alarms.AX_Journal[0][CPT_Message.CV].Message := Message ;
		IN_DataSetFifo_SendSMS.In.Num_tel:=DataSetFifo_ReadSMS.Out.Num;
		IN_DataSetFifo_SendSMS.In.IndexWord:=0;
		IN_DataSetFifo_SendSMS.In.IndexBit:= WORD_TO_SINT(CPT_Message.CV);
		IN_DataSetFifo_SendSMS.A_Add();
		DataSetFifo_ReadSMS.A_Remove();
		
		InStruct.ID := 987;
		InStruct.Message := concat(concat('Le numero de telephone ', IN_DataSetFifo_SendSMS.In.Num_tel), 'a redemarre le PLC') ;
		InStruct.TimeStamp_Act := SYSTEMTIME_TO_STRING(CalLocalTimeStruct);
		//FUN_Alarms_CSV.M_AddAction_FIFO(InStruct := InStruct); // Alarme sur activation du code
		FUN_Alarms_CSV.FIFO.In := InStruct ;
		FUN_Alarms_CSV.FIFO.A_Add() ;
		
	14: // autorisation de couplage
		OpcUa.AllDataWPulse.CmdAutCpl := TRUE;
		
		Message := 'Autorisation de couplage recu';
		FUN_Alarms.AX_Journal[0][CPT_Message.CV].Message := Message ;
		IN_DataSetFifo_SendSMS.In.Num_tel:=DataSetFifo_ReadSMS.Out.Num;
		IN_DataSetFifo_SendSMS.In.IndexWord:=0;
		IN_DataSetFifo_SendSMS.In.IndexBit:= WORD_TO_SINT(CPT_Message.CV);
		IN_DataSetFifo_SendSMS.A_Add();
		DataSetFifo_ReadSMS.A_Remove();
		
		InStruct.ID := 988;
		InStruct.Message := concat(concat('Le numero de telephone ', IN_DataSetFifo_SendSMS.In.Num_tel), 'a envoye une autorisation de couplage') ;
		InStruct.TimeStamp_Act := SYSTEMTIME_TO_STRING(CalLocalTimeStruct);
		//FUN_Alarms_CSV.M_AddAction_FIFO(InStruct := InStruct); // Alarme sur activation du code
		FUN_Alarms_CSV.FIFO.In := InStruct ;
		FUN_Alarms_CSV.FIFO.A_Add() ;
		
	15: // Disconnect order
		OPCUA.AllDataWPulse.CmdDisconnect  := TRUE;
		Message := 'Ordre de decouplage recu';
		FUN_Alarms.AX_Journal[0][CPT_Message.CV].Message := Message ;
		IN_DataSetFifo_SendSMS.In.Num_tel:=DataSetFifo_ReadSMS.Out.Num;
		IN_DataSetFifo_SendSMS.In.IndexWord:=0;
		IN_DataSetFifo_SendSMS.In.IndexBit:= WORD_TO_SINT(CPT_Message.CV);
		IN_DataSetFifo_SendSMS.A_Add();
		DataSetFifo_ReadSMS.A_Remove();
		
		InStruct.ID := 989;
		InStruct.Message := concat(concat('Le numero de telephone ', IN_DataSetFifo_SendSMS.In.Num_tel), ' a fait une demande de decouplage') ;
		InStruct.TimeStamp_Act := SYSTEMTIME_TO_STRING(CalLocalTimeStruct);
		//InStruct
		//FUN_Alarms_CSV.M_AddAction_FIFO(InStruct := InStruct); // Alarme sur activation du code
		FUN_Alarms_CSV.FIFO.In := InStruct ;
		FUN_Alarms_CSV.FIFO.A_Add() ;
	16: // Connect VPN
		OpcUa.AllDataWPulse.CmdStart_Vpn := TRUE;
		Message := 'Starting VPN';
		FUN_Alarms.AX_Journal[0][CPT_Message.CV].Message := Message ;
		IN_DataSetFifo_SendSMS.In.Num_tel:=DataSetFifo_ReadSMS.Out.Num;
		IN_DataSetFifo_SendSMS.In.IndexWord:=0;
		IN_DataSetFifo_SendSMS.In.IndexBit:= WORD_TO_SINT(CPT_Message.CV);
		IN_DataSetFifo_SendSMS.A_Add();
		DataSetFifo_ReadSMS.A_Remove();
		
		InStruct.ID := 990;
		InStruct.Message := concat(concat('Le numero de telephone ', IN_DataSetFifo_SendSMS.In.Num_tel), ' a lance le VPN') ;
		InStruct.TimeStamp_Act := SYSTEMTIME_TO_STRING(CalLocalTimeStruct);
		//InStruct
		//FUN_Alarms_CSV.M_AddAction_FIFO(InStruct := InStruct); // Alarme sur activation du code
		FUN_Alarms_CSV.FIFO.In := InStruct ;
		FUN_Alarms_CSV.FIFO.A_Add() ;
	
	17: // Disconnect VPN
		OpcUa.AllDataWPulse.CmdStop_Vpn := TRUE;
		Message := 'Stopping VPN';
		FUN_Alarms.AX_Journal[0][CPT_Message.CV].Message := Message ;
		IN_DataSetFifo_SendSMS.In.Num_tel:=DataSetFifo_ReadSMS.Out.Num;
		IN_DataSetFifo_SendSMS.In.IndexWord:=0;
		IN_DataSetFifo_SendSMS.In.IndexBit:= WORD_TO_SINT(CPT_Message.CV);
		IN_DataSetFifo_SendSMS.A_Add();
		DataSetFifo_ReadSMS.A_Remove();
		
		InStruct.ID := 991;
		InStruct.Message := concat(concat('Le numero de telephone ', IN_DataSetFifo_SendSMS.In.Num_tel), ' a arrete le VPN') ;
		InStruct.TimeStamp_Act := SYSTEMTIME_TO_STRING(CalLocalTimeStruct);
		//InStruct
		FUN_Alarms_CSV.FIFO.In := InStruct ;
		FUN_Alarms_CSV.FIFO.A_Add() ;
		
	18: // Reboot IPC
		OpcUa.AllDataWPulse.CmdReset_IPC := TRUE;
		Message :='Le PC industriel va redemarer';
		FUN_Alarms.AX_Journal[0][CPT_Message.CV].Message := Message;	
		IN_DataSetFifo_SendSMS.In.Num_tel:=DataSetFifo_ReadSMS.Out.Num;
		IN_DataSetFifo_SendSMS.In.IndexWord:=0;
		IN_DataSetFifo_SendSMS.In.IndexBit:=WORD_TO_SINT(CPT_Message.CV);
		IN_DataSetFifo_SendSMS.A_Add();
		DataSetFifo_ReadSMS.A_Remove();		
END_CASE
END_METHOD

METHOD M_Init : BOOL
VAR_INPUT
END_VAR

VAR

	KK: INT;
	NbrAlarmCodeCSV: INT;
	LL: INT;
	AX_Jou: INT;
END_VAR
END_METHOD

END_PROGRAM

// ---- 00_FunctionsBlocks/Beckhoff/AlarmManagement/FUN_Alarms_CSV.TcPOU
PROGRAM FUN_Alarms_CSV
////////////////// 
// Save Alarms in a CSV File locally. 
//////////////////	
VAR_INPUT
	ParamSeparateur			: STRING := ';';				// Separator for the CSV file
	ParamExtension			: STRING(255) := '.csv';				// File extension
	FIFO					: FB_DBDatasetFifo;	// Buffer that contains all the alarms to be written in the file. 
	
END_VAR
VAR_OUTPUT
	
END_VAR
VAR
	format_string				: FB_Formatstring;
	CalDate						: T_MaxString;
	
	// Alarm management 
		bWriteAlarm				: BOOL;				// Writing CSV File failed 
		TON_WritealarmFile		: TON;				// Tempo to detect error in file creation.  
		
		
	// Data processing 
	MesData		: ServerCSV ;			//  Server info
	CalFileName			: STRING;				// Name of csv file 
	
	//Time Values 
	
	//Test existence file 
	FindFile 			: FB_EnumFindFileEntry ;
	FileInfo			: ST_FindFileEntry;
	bFileOK				: BOOL:= TRUE ;

	//Initial File creation 
	GetHostName			: FB_GetHostName;
	WriteFile			: FB_WriteFile;
	bStartWrite			: BOOL;
	bInitWrite			: BOOL;
	
	//Initial File creation 
	InitLine			: T_MaxString;
	LastInitLine		: T_MaxString;
	WelcomeMessage 		: T_MaxString := 'Daily alarms file';
	ForDay				: T_MaxString := 'for day :';
	ForPlant	 		: T_MaxString := 'for plant : ';
	NewLineVar			: T_MaxString := '$L $00';
	TimeStampVar		: T_MaxString := 'TimeStamp;AlarmsID;Description;Activated;Acknowledged;Level;$L$00';
	MessageInitial		: ARRAY[1..10] OF STRING(255);
	MessageInitial_Null	: ARRAY[1..10] OF STRING(255);
	bInitWriting		: BOOL;
	len_to_write		: INT;
	len_to_add			: INT;

	// Write File
	LineToWrite			: STRING(1000);

	// General variables
		bInit 			: BOOL;
		MesTimeStamp 	: STRING(19);				// Timestamp of the alarm
		bOutCompleted 	: RS;						// Writing file is completed
	
	//TABLEAU
		CalTimeStamp: STRING(255);				// Timestamp formatted

END_VAR

IF NOT bInit THEN
	M_Init();
END_IF

M_AlarmManager();

format_string(
	sFormat := 'ALARMS_%0.2d-%0.2d-%0.2d%s', 
	arg1 := F_WORD(in:=CalLocalTimeStruct.wYear),	arg2 := F_WORD(in:=CalLocalTimeStruct.wMonth),	arg3 := F_WORD(in:=CalLocalTimeStruct.wDay),
	arg4 := F_STRING(in:=ParamExtension),
	sOut => CalFileName
);

format_string(
	sFormat := '%0.2d-%0.2d-%0.2d', 
	arg1 := F_WORD(in:=CalLocalTimeStruct.wYear),	arg2 := F_WORD(in:=CalLocalTimeStruct.wMonth),	arg3 := F_WORD(in:=CalLocalTimeStruct.wDay),
	sOut => CalDate
);

InitLine := concat(str1:=WelcomeMessage, STR2:= concat(str1:=
	ParamSeparateur, str2:=concat(STR1:=ForDay, STR2:=concat(str1:= ParamSeparateur, STR2:= concat(str1:= 
	CalDate,str2:=concat(str1:= ParamSeparateur, str2 := CONCAT(str1:=
	ForPlant,str2:=Concat(str1:=ParamSeparateur, str2:= CONCAT(str1:= GetHostName.sHostName, str2:=ParamSeparateur)
))))))));

IF InitLine <> LastInitLine OR InitLine = '' OR (NOT FindFile.bError AND NOT bFileOK) THEN
	LastInitLine := InitLine;
	bInitWriting := TRUE;
END_IF
		
//Test Existence File
IF FUN_CreateDir_CSV.bDirOk THEN
	FindFile
	(
		sNetId := '',
		sPathName := concat(FUN_CreateDir_CSV.AX_DirNames[2],CalFileName),
		eCmd := eEnumCmd_First,
		bExecute := TRUE,
		tTimeout := T#3S,
		stFindFile => FileInfo
	);
	
 MesData.TimeCreation 	:= FILETIME_TO_SYSTEMTIME(filetime := FileInfo.creationTime);
MesData.TimeModif	 	:= FILETIME_TO_SYSTEMTIME(filetime := FileInfo.lastWriteTime);
	
MesData.FileSize  		:= ULARGE_TO_ULINT(in := FileInfo.fileSize);
	IF NOT FindFile.bBusy THEN
		FindFile(bExecute := FALSE);
		bFileOK := MesData.FileSize > 0 ; 
	END_IF
	
	
	IF NOT FindFile.bBusy AND NOT bFileOK AND bInitWriting THEN
		// je réinitialise les longueurs
		len_to_write := 0;
		MessageInitial := MessageInitial_Null;
		MEMCPY(destAddr := ADR(MessageInitial)+len_to_write, srcAddr := ADR(InitLine), n := len(InitLine));
		len_to_add := len(InitLine);			len_to_write := len_to_write + len_to_add;
		
		MEMCPY(destAddr := ADR(MessageInitial)+len_to_write, srcAddr := ADR(NewLineVar), n := len(NewLineVar));
		len_to_add := len(NewLineVar);			len_to_write := len_to_write + len_to_add;
		
		MEMCPY(destAddr := ADR(MessageInitial)+len_to_write, srcAddr := ADR(TimeStampVar), n := len(TimeStampVar));
		len_to_add := len(TimeStampVar);		len_to_write := len_to_write + len_to_add;
		
		WriteFile
		(
			InStart := TRUE,
			InDirFile := concat(FUN_CreateDir_CSV.AX_DirNames[2], CalFileName),
			InAmsId := '', 
			InPMessage := ADR(MessageInitial),
			InLMessage := len_to_write
		);
		
		IF WriteFile.OutCompleted OR bFileOK THEN
			WriteFile(InStart := FALSE);
		END_IF
	END_IF
	
	
	IF bFileOK AND MesData.FileSize < 100000000 AND fifo.nCount > 0 THEN
		bInitWriting := FALSE;
		fifo.A_Get();	// Unpile the buffer to get the next alarm to write. 
		
		MesTimeStamp := CONCAT(REPLACE(STR1:= left(str := FIFO.Out.TimeStamp_Act, 19), STR2 := ' ', L := 1, P := 11), ' ') ;	// Get Timestamp of the activation or desactivation of the alarm
		ReplaceAll( In_StringTosearch := MesTimeStamp, In_StringToFind := '/', IN_StringToReplace := '-', OUT_StringToSearch => CalTimeStamp);
		
		// Create line content
		LineToWrite := Concat(CalTimeStamp, ParamSeparateur);
		LineToWrite := concat(LineToWrite, Concat(STR1 := UINT_TO_STRING(FIFO.Out.ID) ,ParamSeparateur));
		LineToWrite := concat(LineToWrite, Concat(STR1 := FIFO.Out.Message ,ParamSeparateur));
		LineToWrite := Concat(STR1 := LineToWrite, STR2 := Concat(STR1 := BOOL_TO_STRING( FIFO.Out.Value), STR2 := ParamSeparateur));
		LineToWrite:= Concat(STR1 := LineToWrite, Concat(STR1 := BOOL_TO_STRING( FIFO.Out.Ack), STR2 := ParamSeparateur)); 
		LineToWrite:= Concat(STR1 := LineToWrite, Concat(STR1 := UINT_TO_STRING( FIFO.Out.Alarms_LVL), STR2 := ParamSeparateur)); 
		LineToWrite := Concat(LineToWrite, '$L$00');
		
		// Write File
		WriteFile
		(
			InStart := TRUE,
			InDirFile := concat(FUN_CreateDir_CSV.AX_DirNames[2], CalFileName),
			InAmsId := '', 
			InPMessage := ADR(LineToWrite),
			InLMessage := LEN(LineToWrite)
		);
		IF NOT WriteFile.OutBusy AND NOT WriteFile.OutError AND WriteFile.OutCompleted THEN
			// File has been writen successfully
			fifo.A_Remove();
			WriteFile(InStart := FALSE);
			bWriteAlarm	:= FALSE ;
		ELSIF WriteFile.OutError THEN 
			// In case of writing error, try again to write the alarm. 
			bWriteAlarm	:= TRUE ;
			WriteFile(InStart := FALSE);
		END_IF
	END_IF
END_IF

METHOD M_AlarmManager
VAR

	FB_AlarmCodeManager			: FB_AlarmCodeManager ;

END_VAR

TON_WritealarmFile(IN:= NOT bFileOK  , PT:= T#10S  ) ;


// ALARM CODE //
	FB_AlarmCodeManager(
		bAlarm1			:= bWriteAlarm	  ,				// Write CSV Alarm
		bAlarm2			:= fifo.bOverwrite   ,			// Overflow buffer
		bAlarm3			:= TON_WritealarmFile.Q   ,		// Can not create CSV Alarm file 
		bAlarm4			:= FALSE	 ,					//
		bAlarm5			:= FALSE	,					// 
		bAlarm6			:= FALSE,									//
		bAlarm7			:= FALSE,                                   //
		bAlarm8			:= FALSE,                                   //
		bAlarm9			:= FALSE,                                   //
		bAlarm10		:= FALSE,                                   //
		bAlarm11		:= FALSE,									//
		bAlarm12		:= FALSE,                                   //
		bAlarm13		:= FALSE,                                   //
		bAlarm14		:= FALSE,                                   //
		bAlarm15		:= FALSE,                                   //
		wAlarmCode		=>MesData.MesAlarmCode);
END_METHOD

METHOD M_Init

VAR
	LL	: SINT;
	KK 	: SINT;
	InStruct : ST_ValuesAlarms;
END_VAR
// Create a first alarm after new code activation or PLC restart
//	FIFO.A_Get();
//	FIFO.A_Remove();
	bInit := TRUE;


	GetHostName(bExecute := FALSE);
	GetHostName(bExecute := TRUE);
END_METHOD

END_PROGRAM

// ---- 00_FunctionsBlocks/Beckhoff/Communication/Mail/FUN_SendMail.TcPOU
PROGRAM FUN_SendMail
////////////////// 
// Send Alarms by mails. 
//////////////////

VAR_INPUT
	ParamTempoTimeout				: TIME := T#20S;		(* (s) Tempo before timeout. *)
	IN_Directory 					: T_maxstring := 'C:\TwinCAT\Functions\Annex_Fonctions\SendEmail\';	// Directory of the SMTP.Exe file. 
	IN_Reset_OPC					: BOOL;					// Reset Mail server and alarms. 
	IN_Restart_Service_OPC			: BOOL;					// Restart SMTP services. 
	IN_ChangePhoneMailInfos_OPC		: BOOL;					// Change users Info (mails, name, Lvl, ... ) 
	FIFO							: FB_DBDatasetFifo;		// Buffer of the alarmes). 
	
END_VAR

VAR_OUTPUT
	OUT_Completed					: BOOL;		// Juste un trig pour dire que c'est fini. Written by the SMTP.Exe
	OUT_Error						: BOOL;		// Tant qu'il y a une erreur. Written by the SMTP.exe
	OUT_Busy						: BOOL;		// Envoi en cours. 
	OUT_NbMailSent 					: UINT;	// Number of mail being sent. 
END_VAR

VAR PERSISTENT
	AX_MailAddr						: ARRAY[1..CstNbUser] OF STRING(255);	//Contient tous les numéros des utilisateurs
	AX_Subscribed					: ARRAY[1..CstNbUser] OF BOOL		;	// List of subscription. 
	AX_NomUtili						: ARRAY[1..CstNbUser] OF STRING(50)	;	// List of user names. 
	AX_User_LVL						: ARRAY[1..CstNbUser] OF WORD;			//Contient tous les niveau d'adhésion des utilisateurs.
END_VAR

VAR_INPUT PERSISTENT
	ParamTempoRetry					: TIME := T#1M;  (* (s) Tempo before send email retry *) 
	ParamNetID						: STRING :='' ; (* AMS Net ID where the SMTP.exe file is stored *)
END_VAR

VAR

	// M_AlarmManager 
	MesData			: ServerMail;
	RS_AlarmDestinator		: RS;
	
	// M_Write Param	
	bAlarmNoDestinator		: BOOL;
	bSendMail				: BOOL;
	
	bWriteParam				: BOOL;
	Body					: T_MaxString;
	MailAddr				: T_MaxString;
	MesTimeStamp			: STRING(17);	
	CalTimeStamp			: STRING(255);

	//M_Send
	SendMail				: NT_StartProcess;
	
	//M_OPC
	Trig_OPC				: R_TRIG;
	RS_OPC					: RS;
	Trig_Reset				: R_TRIG;

	KK						: UINT;
	NbDest					: INT;
	TON_Retry				: TON;
	Old_Count				: UDINT;
	R_TRIG_Retry			: R_TRIG;
	
END_VAR

M_AlarmManager();
M_OPC();
M_Evaluate();

IF IN_Reset_OPC THEN
	M_Reset();
END_IF
TON_Retry(IN := Old_Count = fifo.nCount AND NOT R_TRIG_Retry.Q, pt := ParamTempoRetry);

R_TRIG_Retry(clk := TON_Retry.Q);
IF old_count <> fifo.nCount THEN
	Old_Count := fifo.nCount;
END_IF
bWriteParam := fifo.nCount > 0; 	// if the buffer is not empty, send mail. 
fifo.A_Get();	// Get the next alarm to send. 

MesTimeStamp := CONCAT(REPLACE(STR1:= left(str := FIFO.Out.TimeStamp_Act, 16), STR2 := ' ', L := 1, P := 11), ' ') ;
ReplaceAll( In_StringTosearch := MesTimeStamp, In_StringToFind := '/', IN_StringToReplace := '-', OUT_StringToSearch => CalTimeStamp);

Body := concat(left(FIFO.Out.Message, 125),SEL(FIFO.Out.Value, ' : Desactive"',' : Active"')) ; 
Body := concat( STR1:= UINT_TO_STRING(FIFO.Out.ID) , STR2:= concat(STR1:=' ,' , STR2:=Body )) ; 
Body := concat( STR1:= 'ID:' , STR2:=Body ) ; 
Body := concat('"', Concat(CalTimeStamp,Body));


